				MB_BitStato[100]:=ModBus.MB_MASTER.ReceiveBuffer.Data[3].0; (*Vedi Tabella *)
				MB_BitStato[101]:=ModBus.MB_MASTER.ReceiveBuffer.Data[3].1; (*Vedi Tabella *)
				MB_BitStato[102]:=ModBus.MB_MASTER.ReceiveBuffer.Data[3].2; (*Vedi Tabella *)
				MB_BitStato[103]:=ModBus.MB_MASTER.ReceiveBuffer.Data[3].3; (*Vedi Tabella *)
				MB_BitStato[104]:=ModBus.MB_MASTER.ReceiveBuffer.Data[3].4; (*Vedi Tabella *)
				MB_BitStato[105]:=ModBus.MB_MASTER.ReceiveBuffer.Data[3].5; (*Vedi Tabella *)
				MB_BitStato[106]:=ModBus.MB_MASTER.ReceiveBuffer.Data[3].6; (*Vedi Tabella *)
				MB_BitStato[107]:=ModBus.MB_MASTER.ReceiveBuffer.Data[3].7; (*Vedi Tabella *)
				MB_BitStato[108]:=ModBus.MB_MASTER.ReceiveBuffer.Data[4].0; (*Vedi Tabella *)
				MB_BitStato[109]:=ModBus.MB_MASTER.ReceiveBuffer.Data[4].1; (*Vedi Tabella *)
				MB_BitStato[110]:=ModBus.MB_MASTER.ReceiveBuffer.Data[4].2; (*Vedi Tabella *)
				MB_BitStato[111]:=ModBus.MB_MASTER.ReceiveBuffer.Data[4].3; (*Vedi Tabella *)
				MB_BitStato[112]:=ModBus.MB_MASTER.ReceiveBuffer.Data[4].4; (*Vedi Tabella *)
				MB_BitStato[113]:=ModBus.MB_MASTER.ReceiveBuffer.Data[4].5; (*Vedi Tabella *)
				MB_BitStato[114]:=ModBus.MB_MASTER.ReceiveBuffer.Data[4].6; (*Vedi Tabella *)
				MB_BitStato[115]:=ModBus.MB_MASTER.ReceiveBuffer.Data[4].7; (*Vedi Tabella *)
				MB_BitStato[116]:=ModBus.MB_MASTER.ReceiveBuffer.Data[5].0; (*Vedi Tabella *)
				MB_BitStato[117]:=ModBus.MB_MASTER.ReceiveBuffer.Data[5].1; (*Vedi Tabella *)
				MB_BitStato[118]:=ModBus.MB_MASTER.ReceiveBuffer.Data[5].2; (*Vedi Tabella *)
				MB_BitStato[119]:=ModBus.MB_MASTER.ReceiveBuffer.Data[5].3; (*Vedi Tabella *)
				MB_BitStato[120]:=ModBus.MB_MASTER.ReceiveBuffer.Data[5].4; (*Vedi Tabella *)
				MB_BitStato[121]:=ModBus.MB_MASTER.ReceiveBuffer.Data[5].5; (*Vedi Tabella *)
				MB_BitStato[122]:=ModBus.MB_MASTER.ReceiveBuffer.Data[5].6; (*Vedi Tabella *)
				MB_BitStato[123]:=ModBus.MB_MASTER.ReceiveBuffer.Data[5].7; (*Vedi Tabella *)
				MB_BitStato[124]:=ModBus.MB_MASTER.ReceiveBuffer.Data[6].0; (*Vedi Tabella *)
				MB_BitStato[125]:=ModBus.MB_MASTER.ReceiveBuffer.Data[6].1; (*Vedi Tabella *)
				MB_BitStato[126]:=ModBus.MB_MASTER.ReceiveBuffer.Data[6].2; (*Vedi Tabella *)
				MB_BitStato[127]:=ModBus.MB_MASTER.ReceiveBuffer.Data[6].3; (*Vedi Tabella *)
				MB_BitStato[128]:=ModBus.MB_MASTER.ReceiveBuffer.Data[6].4; (*Vedi Tabella *)
				MB_BitStato[129]:=ModBus.MB_MASTER.ReceiveBuffer.Data[6].5; (*Vedi Tabella *)
				MB_BitStato[130]:=ModBus.MB_MASTER.ReceiveBuffer.Data[6].6; (*Vedi Tabella *)
				MB_BitStato[131]:=ModBus.MB_MASTER.ReceiveBuffer.Data[6].7; (*Vedi Tabella *)
				MB_BitStato[132]:=ModBus.MB_MASTER.ReceiveBuffer.Data[7].0; (*Vedi Tabella *)
				MB_BitStato[133]:=ModBus.MB_MASTER.ReceiveBuffer.Data[7].1; (*Vedi Tabella *)
				MB_BitStato[134]:=ModBus.MB_MASTER.ReceiveBuffer.Data[7].2; (*Vedi Tabella *)
				MB_BitStato[135]:=ModBus.MB_MASTER.ReceiveBuffer.Data[7].3; (*Vedi Tabella *)
				MB_BitStato[136]:=ModBus.MB_MASTER.ReceiveBuffer.Data[7].4; (*Vedi Tabella *)
				MB_BitStato[137]:=ModBus.MB_MASTER.ReceiveBuffer.Data[7].5; (*Vedi Tabella *)
				MB_BitStato[138]:=ModBus.MB_MASTER.ReceiveBuffer.Data[7].6; (*Vedi Tabella *)
				MB_BitStato[139]:=ModBus.MB_MASTER.ReceiveBuffer.Data[7].7; (*Vedi Tabella *)
				MB_BitStato[140]:=ModBus.MB_MASTER.ReceiveBuffer.Data[8].0; (*Vedi Tabella *)
				MB_BitStato[141]:=ModBus.MB_MASTER.ReceiveBuffer.Data[8].1; (*Vedi Tabella *)
				MB_BitStato[142]:=ModBus.MB_MASTER.ReceiveBuffer.Data[8].2; (*Vedi Tabella *)
				MB_BitStato[143]:=ModBus.MB_MASTER.ReceiveBuffer.Data[8].3; (*Vedi Tabella *)
				MB_BitStato[144]:=ModBus.MB_MASTER.ReceiveBuffer.Data[8].4; (*Vedi Tabella *)
				MB_BitStato[145]:=ModBus.MB_MASTER.ReceiveBuffer.Data[8].5; (*Vedi Tabella *)
				MB_BitStato[146]:=ModBus.MB_MASTER.ReceiveBuffer.Data[8].6; (*Vedi Tabella *)
				MB_BitStato[147]:=ModBus.MB_MASTER.ReceiveBuffer.Data[8].7; (*Vedi Tabella *)
				MB_BitStato[148]:=ModBus.MB_MASTER.ReceiveBuffer.Data[9].0; (*Vedi Tabella *)
				MB_BitStato[149]:=ModBus.MB_MASTER.ReceiveBuffer.Data[9].1; (*Vedi Tabella *)
				MB_BitStato[150]:=ModBus.MB_MASTER.ReceiveBuffer.Data[9].2; (*Vedi Tabella *)
				MB_BitStato[151]:=ModBus.MB_MASTER.ReceiveBuffer.Data[9].3; (*Vedi Tabella *)
				MB_BitStato[152]:=ModBus.MB_MASTER.ReceiveBuffer.Data[9].4; (*Vedi Tabella *)
				MB_BitStato[153]:=ModBus.MB_MASTER.ReceiveBuffer.Data[9].5; (*Vedi Tabella *)
				MB_BitStato[154]:=ModBus.MB_MASTER.ReceiveBuffer.Data[9].6; (*Vedi Tabella *)
				MB_BitStato[155]:=ModBus.MB_MASTER.ReceiveBuffer.Data[9].7; (*Vedi Tabella *)
				MB_BitStato[156]:=ModBus.MB_MASTER.ReceiveBuffer.Data[10].0; (*Vedi Tabella *)
				MB_BitStato[157]:=ModBus.MB_MASTER.ReceiveBuffer.Data[10].1; (*Vedi Tabella *)
				MB_BitStato[158]:=ModBus.MB_MASTER.ReceiveBuffer.Data[10].2; (*Vedi Tabella *)
				MB_BitStato[159]:=ModBus.MB_MASTER.ReceiveBuffer.Data[10].3; (*Vedi Tabella *)
				MB_BitStato[160]:=ModBus.MB_MASTER.ReceiveBuffer.Data[10].4; (*Vedi Tabella *)
				MB_BitStato[161]:=ModBus.MB_MASTER.ReceiveBuffer.Data[10].5; (*Vedi Tabella *)
				MB_BitStato[162]:=ModBus.MB_MASTER.ReceiveBuffer.Data[10].6; (*Vedi Tabella *)
				MB_BitStato[163]:=ModBus.MB_MASTER.ReceiveBuffer.Data[10].7; (*Vedi Tabella *)
				MB_BitStato[164]:=ModBus.MB_MASTER.ReceiveBuffer.Data[11].0; (*Vedi Tabella *)
				MB_BitStato[165]:=ModBus.MB_MASTER.ReceiveBuffer.Data[11].1; (*Vedi Tabella *)
				MB_BitStato[166]:=ModBus.MB_MASTER.ReceiveBuffer.Data[11].2; (*Vedi Tabella *)
				MB_BitStato[167]:=ModBus.MB_MASTER.ReceiveBuffer.Data[11].3; (*Vedi Tabella *)
				MB_BitStato[168]:=ModBus.MB_MASTER.ReceiveBuffer.Data[11].4; (*Vedi Tabella *)
				MB_BitStato[169]:=ModBus.MB_MASTER.ReceiveBuffer.Data[11].5; (*Vedi Tabella *)
				MB_BitStato[170]:=ModBus.MB_MASTER.ReceiveBuffer.Data[11].6; (*Vedi Tabella *)
				MB_BitStato[171]:=ModBus.MB_MASTER.ReceiveBuffer.Data[11].7; (*Vedi Tabella *)
				MB_BitStato[172]:=ModBus.MB_MASTER.ReceiveBuffer.Data[12].0; (*Vedi Tabella *)
				MB_BitStato[173]:=ModBus.MB_MASTER.ReceiveBuffer.Data[12].1; (*Vedi Tabella *)
				MB_BitStato[174]:=ModBus.MB_MASTER.ReceiveBuffer.Data[12].2; (*Vedi Tabella *)
				MB_BitStato[175]:=ModBus.MB_MASTER.ReceiveBuffer.Data[12].3; (*Vedi Tabella *)
				MB_BitStato[176]:=ModBus.MB_MASTER.ReceiveBuffer.Data[12].4; (*Vedi Tabella *)
				MB_BitStato[177]:=ModBus.MB_MASTER.ReceiveBuffer.Data[12].5; (*Vedi Tabella *)
				MB_BitStato[178]:=ModBus.MB_MASTER.ReceiveBuffer.Data[12].6; (*Vedi Tabella *)
				MB_BitStato[179]:=ModBus.MB_MASTER.ReceiveBuffer.Data[12].7; (*Vedi Tabella *)
				MB_BitStato[180]:=ModBus.MB_MASTER.ReceiveBuffer.Data[13].0; (*Vedi Tabella *)
				MB_BitStato[181]:=ModBus.MB_MASTER.ReceiveBuffer.Data[13].1; (*Vedi Tabella *)
				MB_BitStato[182]:=ModBus.MB_MASTER.ReceiveBuffer.Data[13].2; (*Vedi Tabella *)
				MB_BitStato[183]:=ModBus.MB_MASTER.ReceiveBuffer.Data[13].3; (*Vedi Tabella *)
				MB_BitStato[184]:=ModBus.MB_MASTER.ReceiveBuffer.Data[13].4; (*Vedi Tabella *)
				MB_BitStato[185]:=ModBus.MB_MASTER.ReceiveBuffer.Data[13].5; (*Vedi Tabella *)
				MB_BitStato[186]:=ModBus.MB_MASTER.ReceiveBuffer.Data[13].6; (*Vedi Tabella *)
				MB_BitStato[187]:=ModBus.MB_MASTER.ReceiveBuffer.Data[13].7; (*Vedi Tabella *)
				MB_BitStato[188]:=ModBus.MB_MASTER.ReceiveBuffer.Data[13].0; (*Vedi Tabella *)
				MB_BitStato[189]:=ModBus.MB_MASTER.ReceiveBuffer.Data[13].1; (*Vedi Tabella *)
				MB_BitStato[190]:=ModBus.MB_MASTER.ReceiveBuffer.Data[13].2; (*Vedi Tabella *)
				MB_BitStato[191]:=ModBus.MB_MASTER.ReceiveBuffer.Data[13].3; (*Vedi Tabella *)
				MB_BitStato[192]:=ModBus.MB_MASTER.ReceiveBuffer.Data[13].4; (*Vedi Tabella *)
				MB_BitStato[193]:=ModBus.MB_MASTER.ReceiveBuffer.Data[13].5; (*Vedi Tabella *)
				MB_BitStato[194]:=ModBus.MB_MASTER.ReceiveBuffer.Data[13].6; (*Vedi Tabella *)
				MB_BitStato[195]:=ModBus.MB_MASTER.ReceiveBuffer.Data[13].7; (*Vedi Tabella *)
				MB_BitStato[196]:=ModBus.MB_MASTER.ReceiveBuffer.Data[14].0; (*Vedi Tabella *)
				MB_BitStato[197]:=ModBus.MB_MASTER.ReceiveBuffer.Data[14].1; (*Vedi Tabella *)
				MB_BitStato[198]:=ModBus.MB_MASTER.ReceiveBuffer.Data[14].2; (*Vedi Tabella *)
				MB_BitStato[199]:=ModBus.MB_MASTER.ReceiveBuffer.Data[14].3; (*Vedi Tabella *)


				state:=290;

			END_IF
		END_IF




		290:    (* Scrittura BOOL - COIL o WORD *)
		IF NOT ModBus.MB_Start THEN
			IF ModBus.MB_MASTER.MB_Error<>0 THEN (*OR ModBus.MB_MASTER.MB_Error<>0 THEN*)
				state := 300;
			ELSE
				IF ScriviDato THEN
					IF ScriviCoil THEN
						Modbus.MB_Query.FunctionCode := 5;
					ELSE
						Modbus.MB_Query.FunctionCode := 6;
					END_IF
					Modbus.MB_Query.SlaveAddress := Address;
					ModBus.MB_Query.Write_StartAddress := IndirizzoDaScrivere;
					ModBus.MB_Query.Write_Quantity :=1;
					ModBus.MB_Query.Write_Data[0] := DatoDaScrivere;
					ModBus.MB_Start := TRUE;
						IF ScriviCoil THEN
							IF 	MB_BitStato[IndirizzoDaScrivere]=WORD_TO_BOOL(DatoDaScrivere-1) THEN
								ScriviDato:=FALSE;
							END_IF
						ELSE
							IF 	MB_RegistriLetti[IndirizzoDaScrivere]=DatoDaScrivere THEN
								ScriviDato:=FALSE;
							END_IF
						END_IF
					state := 295;
				ELSE
					state := 295;
				END_IF
			END_IF
		END_IF




		295:
		IF NOT ModBus.MB_Start THEN
			IF ModBus.MB_MASTER.MB_Error<>0 THEN (*OR ModBus.MB_MASTER.MB_Error<>0 THEN*)
				state := 300;
			ELSE
				IF fModbusAlr THEN fModbusAlr := FALSE; END_IF
				NodoDaInterrogareChiller:=Address+1;
				InibiscoModbusChiller:=FALSE;
				retryErr := 0;
				retry := 0;
				state := 0;
					IF fModbusAlr=FALSE AND ErroreComuModBus=TRUE THEN
						LogEv(EL_Log,EO_CHI,ID,62,'ComunicazioneModBus_OK');
						ErroreComuModBus := FALSE;
				(*	WarningCtr := SEL(WarningCtr=0, WarningCtr-1, 0); *)
					END_IF


			END_IF
		END_IF



	(**** CHECK MODBUS ERROR ****)
	300: 	(* Release MODBUS *)
			InibiscoModbusChiller:=FALSE;
			(* Retries *)
			retry:=retry+1;
			IF retry>3 THEN
				retry:=0;

				(* Verify if slave is dead *)
				IF retryErr < retryErrMaX THEN
					retryErr := retryErr + 1;
				ELSE
					fModbusAlr := TRUE;
					(* Verify ModBus error	*)

					IF fModbusAlr AND ErroreComuModBus=FALSE THEN
						LogEv(EL_Alarm,EO_CHI,ID,61,CONCAT('ErroreModbus_',INT_TO_STRING(ModBus.MB_MASTER.MB_Error)));
						ErroreComuModBus := TRUE;
					END_IF
				END_IF

				END_IF
			Refresh_Now := FALSE;
			NodoDaInterrogareChiller:=Address+1;
			state:=0;
END_CASE




(* Controllo Time Out Ciclo ModBus *)

TimeOutModBus(In:=state<>0,PT:=t#30s);
IF TimeOutModBus.Q THEN
	State:=0;
	Refresh_Now:=TRUE;  (* Rilancio la lettura del nodo *)
	IF MODBUS.MB_Lock=TRUE THEN MODBUS.MB_Lock:=FALSE;END_IF
	IF InibiscoModbusChiller=TRUE THEN InibiscoModbusChiller:=FALSE;END_IF
END_IF
END_ACTION

(* POU Utils Functions/TONOF, ST *)
FUNCTION_BLOCK TONOF
VAR_INPUT
	IN		: BOOL;
	PT_ON	: TIME; (* time to pass, before OUT is set *)
	PT_OF	: TIME; (* time to pass, before OUT is reset *)
END_VAR
VAR_OUTPUT
	OUT		: BOOL;
END_VAR
VAR
	timer	: TON;
END_VAR
IF IN<>OUT THEN
	timer(IN:=TRUE,PT:=SEL(IN,PT_OF,PT_ON));
	IF timer.Q THEN OUT:=IN; END_IF
ELSE
	timer(IN:=FALSE);
END_IF
END_FUNCTION_BLOCK

(* POU Plant_Objects/obj_MODBUS_TRENDCOIN_01, ST *)
FUNCTION_BLOCK obj_MODBUS_TRENDCOIN_01
VAR CONSTANT

	TimeOutModBus: TON;


END_VAR
VAR_INPUT
	ID			:	BYTE;
	Address		:	BYTE;
	(* Modbus *)
	Refresh_Now	:	BOOL;			(* Richiesta di lettura stato macchina Immediata  *)
	retryErrMax	:	BYTE := 2;

	IndirizzoDaScrivere: WORD;
	DatoDaScrivere: INT;
	ScriviDato: BOOL;
	ScriviCoil: BOOL;

(* Variabili da scrivere nel parametri Trend *)

(*	EnScrittura		:ARRAY [0..15] OF	FLT_EVENT; *)

	ControlMode_UTA01:BOOL;     (* 0 = controllato in manuale ; 1 = controllato col Crono *)
	ControlMode_UTA02:BOOL;
	ControlMode_UTA03:BOOL;
	ControlMode_UTA04:BOOL;
	ControlMode_UTA05:BOOL;
	ControlMode_UTA06:BOOL;
	ControlMode_UTA07:BOOL;
	ControlMode_UTA08:BOOL;
	ControlMode_UTA09:BOOL;
	ControlMode_UTA10:BOOL;
	ControlMode_UTA12:BOOL;
	ControlMode_UTA13:BOOL;

	ScriviRUN_UTA01:BOOL;
	ScriviRUN_UTA02:BOOL;
	ScriviRUN_UTA03:BOOL;
	ScriviRUN_UTA04:BOOL;
	ScriviRUN_UTA05:BOOL;
	ScriviRUN_UTA06:BOOL;
	ScriviRUN_UTA07:BOOL;
	ScriviRUN_UTA08:BOOL;
	ScriviRUN_UTA09:BOOL;
	ScriviRUN_UTA10:BOOL;
	ScriviRUN_UTA12:BOOL;
	ScriviRUN_UTA13:BOOL;

	ScriviSP_UTA01:INT;
	ScriviSP_UTA02:INT;
	ScriviSP_UTA03:INT;
	ScriviSP_UTA04:INT;
	ScriviSP_UTA05:INT;
	ScriviSP_UTA06:INT;
	ScriviSP_UTA07:INT;
	ScriviSP_UTA08:INT;
	ScriviSP_UTA09:INT;
	ScriviSP_UTA10:INT;
	ScriviSP_UTA12:INT;
	ScriviSP_UTA13:INT;


END_VAR
VAR_IN_OUT
	ModBus		:obj_MODBUS;

END_VAR
VAR_OUTPUT
	Status_Log	:	WORD;
	Status_Vis	:	DWORD;
END_VAR
VAR

	state		:	INT;
	retry		:	BYTE;
	retryErr	:	BYTE;
	ReadTmr		:	TON := (PT:=T#5s);
	fModbusAlr:BOOL;

(*	retry_write	:	BYTE;
	fWriteStatus:	BOOL;
	fWriteMode	:	BOOL;
	fWriteReset	:	BOOL; *)

	x: INT;

	VerificaFuctionCode: INT;
	VerificaNodoLetto: INT;
	ErroreComuModBus: BOOL;
	IndiceErrore: BYTE;

	MB_BitStato: ARRAY [0..450] OF BOOL;
	MB_RegistriLetti: ARRAY [0..450] OF INT;
	MB_RegistriHoldingLetti: ARRAY [0..170] OF INT;
	MB_BitStatoCoil: ARRAY [0..100] OF BOOL;




	AddressRead: BYTE;
	index: BYTE;
	indexErr: BYTE;


	Read_StartAddress: INT;
	Read_Quantity: BYTE;
	IndiceMBLettura: INT;
	IndiceMBLetto: INT;



	test_Address: INT;
	Test_ScriviCoil: BOOL;
	test_Write: WORD;
	ScriviMB: BOOL;



	AddressDaScrivere: INT;


	temp :STRING(255);
	tempRaw		: ARRAY [0..MAX_SEND_TCP_CLIENT] OF BYTE;
	tempRawLen :DINT;
	longString:STRING(800);


END_VAR
(*
	EnScrittura[1](IN:=Abilita_UTA01);
	ScriviRUN_UTA01:=EnScrittura[1].EVH;
	ScriviRUN_UTA01:=EnScrittura[1].EVL;

	EnScrittura[2](IN:=Abilita_UTA02);
	ScriviRUN_UTA02:=EnScrittura[2].EVH;
	ScriviRUN_UTA02:=EnScrittura[2].EVL;

	EnScrittura[3](IN:=Abilita_UTA03);
	ScriviRUN_UTA03:=EnScrittura[3].EVH;
	ScriviRUN_UTA03:=EnScrittura[3].EVL;

	EnScrittura[4](IN:=Abilita_UTA04);
	ScriviRUN_UTA04:=EnScrittura[4].EVH;
	ScriviRUN_UTA04:=EnScrittura[4].EVL;

	EnScrittura[4](IN:=Abilita_UTA04);
	ScriviRUN_UTA04:=EnScrittura[4].EVH;
	ScriviRUN_UTA04:=EnScrittura[4].EVL;

	EnScrittura[5](IN:=Abilita_UTA05);
	ScriviRUN_UTA05:=EnScrittura[5].EVH;
	ScriviRUN_UTA05:=EnScrittura[5].EVL;

	EnScrittura[6](IN:=Abilita_UTA06);
	ScriviRUN_UTA06:=EnScrittura[6].EVH;
	ScriviRUN_UTA06:=EnScrittura[6].EVL;

	EnScrittura[7](IN:=Abilita_UTA07);
	ScriviRUN_UTA07:=EnScrittura[7].EVH;
	ScriviRUN_UTA07:=EnScrittura[7].EVL;

	EnScrittura[8](IN:=Abilita_UTA08);
	ScriviRUN_UTA08:=EnScrittura[8].EVH;
	ScriviRUN_UTA08:=EnScrittura[8].EVL;

	EnScrittura[9](IN:=Abilita_UTA09);
	ScriviRUN_UTA09:=EnScrittura[9].EVH;
	ScriviRUN_UTA09:=EnScrittura[9].EVL;

	EnScrittura[10](IN:=Abilita_UTA10);
	ScriviRUN_UTA10:=EnScrittura[10].EVH;
	ScriviRUN_UTA10:=EnScrittura[10].EVL;

(*	EnScrittura[11](IN:=Abilita_UTA11);
	ScriviRUN_UTA11:=EnScrittura[11].EVH;
	ScriviRUN_UTA11:=EnScrittura[11].EVL; *)

	EnScrittura[12](IN:=Abilita_UTA12);
	ScriviRUN_UTA12:=EnScrittura[12].EVH;
	ScriviRUN_UTA12:=EnScrittura[12].EVL;

	EnScrittura[13](IN:=Abilita_UTA13);
	ScriviRUN_UTA13:=EnScrittura[13].EVH;
	ScriviRUN_UTA13:=EnScrittura[13].EVL;
*)





(* Call ModBus state machine *)
Stm();

(* Check alarm	*)




(* Seganalzione stato Frigorifero  *)
IF ErroreComuModBus THEN
		Status_Log:=2; Status_Vis:=16#2020F0;
(*	ELSIF Warning OR Warning2 THEN
		Status_Log:=1; Status_Vis:=16#20F0F0; *)
    ELSE
		Status_Log:=0;
		Status_Vis:=16#006000;
END_IF
END_FUNCTION_BLOCK
ACTION AddLogData:
Logger.s1:=INSERT('&POOL=',BYTE_TO_STRING(ID),5);
IF ID<10 THEN Logger.s1:=INSERT(Logger.s1,'0',5); END_IF


(* inizializzo stringa da loggare **)
FOR tempRawLen:=0 TO MAX_SEND_TCP_CLIENT DO
                tempRaw[tempRawLen]:=0;
END_FOR

tempRawLen:=0;


temp:=Logger.s1;
ADDSTRING(ADR(tempRaw), ADR(temp), tempRawLen);

(* Sparo i COIL **)
FOR x:= 1 TO 65 DO
	temp:=CONCAT(SEL(MB_BitStatoCoil[x],'0','1'),';');
	ADDSTRING(ADR(tempRaw), ADR(temp), tempRawLen);
END_FOR

(* Sparo gli ingressi Digitali **)
FOR x:= 1 TO 358 DO
	temp:=CONCAT(SEL(MB_BitStato[x],'0','1'),';');
	ADDSTRING(ADR(tempRaw), ADR(temp), tempRawLen);
END_FOR

(* Sparo gli HOLDING **)
FOR x:= 1 TO 168 DO
	temp:=CONCAT(INT_TO_STRING(MB_RegistriHoldingLetti[x]),';');
	ADDSTRING(ADR(tempRaw), ADR(temp), tempRawLen);
END_FOR

(* Sparo gli integer **)
FOR x:= 1 TO 283 DO
	temp:=CONCAT(INT_TO_STRING(MB_RegistriLetti[x]),';');
	ADDSTRING(ADR(tempRaw), ADR(temp), tempRawLen);
END_FOR

	temp:=(INT_TO_STRING(MB_RegistriLetti[284]));
	ADDSTRING(ADR(tempRaw), ADR(temp), tempRawLen);

ADDSTRING(ADR(Logger.TData), ADR(tempRaw), Logger.TLen);
END_ACTION
ACTION Stm:
CASE state OF
	0:	(* Refresh time manager *)
		ReadTmr(IN:=NOT ReadTmr.Q);
		(*A tempo interrogo il nodo sempre che non ci sia qualcuno che lo sta interrogando in quel momento *)

		IF (ReadTmr.Q AND NodoDaInterrogareMB1=Address )OR Refresh_Now AND NOT InibiscoModbusMB1 THEN
			state := 10;
			ReadTmr.PT := T#10s;  (* moreno *)
			Refresh_Now := FALSE;
			InibiscoModbusMB1 := TRUE;
		END_IF

	(**** Leggo le Analogiche a Disposzione  ****)

	10:	(* richiedo lettura di tutti gli Input Register   *)

		Modbus.MB_Query.SlaveAddress := Address;
		Modbus.MB_Query.FunctionCode := 4;
		Read_StartAddress := 0 ;			(* richiedo lettura altri Parametri *)
		Read_Quantity := 20;
		ModBus.MB_Start := TRUE;
		state := 20;


	20:
		ModBus.MB_Query.Read_StartAddress := 0 ;			(* richiedo lettura altri Parametri *)
		ModBus.MB_Query.Read_Quantity := 20;
		ModBus.MB_Start := TRUE;
		Read_StartAddress := 0 ;
		state := 30;



	30:	(* Risposta all'interrogazione *)
		IF NOT ModBus.MB_Start   THEN
			VerificaFuctionCode:=ModBus.MB_Resp.FunctionCode;
			VerificaNodoLetto:=ModBus.MB_Resp.SlaveAddress;

			IF ModBus.MB_MASTER.MB_Error<>0 THEN
				state := 300;
			ELSE

				FOR x:= 0 TO ModBus.MB_Query.Read_Quantity DO
					MB_RegistriLetti[Read_StartAddress+x ] := ModBus.MB_Resp.Data[x];   	(* Vedi tabella *)
				END_FOR

			ModBus.MB_Query.Read_StartAddress := 20 ;			(* richiedo lettura altri Parametri *)
			ModBus.MB_Query.Read_Quantity := 20;
			ModBus.MB_Start := TRUE;
			Read_StartAddress := 20 ;
			state := 31;
			END_IF
		END_IF


	31:	(* Risposta all'interrogazione *)
		IF NOT ModBus.MB_Start   THEN
			VerificaFuctionCode:=ModBus.MB_Resp.FunctionCode;
			VerificaNodoLetto:=ModBus.MB_Resp.SlaveAddress;

			IF ModBus.MB_MASTER.MB_Error<>0 THEN
				state := 300;
			ELSE

				FOR x:= 0 TO ModBus.MB_Query.Read_Quantity DO
					MB_RegistriLetti[Read_StartAddress+x ] := ModBus.MB_Resp.Data[x];   	(* Vedi tabella *)
				END_FOR

			ModBus.MB_Query.Read_StartAddress := 40 ;			(* richiedo lettura altri Parametri *)
			ModBus.MB_Query.Read_Quantity := 20;
			ModBus.MB_Start := TRUE;
			Read_StartAddress := 40 ;
			state := 32;
			END_IF
		END_IF



	32:	(* Risposta all'interrogazione *)
		IF NOT ModBus.MB_Start   THEN
			VerificaFuctionCode:=ModBus.MB_Resp.FunctionCode;
			VerificaNodoLetto:=ModBus.MB_Resp.SlaveAddress;

			IF ModBus.MB_MASTER.MB_Error<>0 THEN
				state := 300;
			ELSE

				FOR x:= 0 TO ModBus.MB_Query.Read_Quantity DO
					MB_RegistriLetti[Read_StartAddress+x ] := ModBus.MB_Resp.Data[x];   	(* Vedi tabella *)
				END_FOR

			ModBus.MB_Query.Read_StartAddress := 60 ;			(* richiedo lettura altri Parametri *)
			ModBus.MB_Query.Read_Quantity := 20;
			ModBus.MB_Start := TRUE;
			Read_StartAddress := 60 ;
			state := 33;
			END_IF
		END_IF

	33:	(* Risposta all'interrogazione *)
		IF NOT ModBus.MB_Start   THEN
			VerificaFuctionCode:=ModBus.MB_Resp.FunctionCode;
			VerificaNodoLetto:=ModBus.MB_Resp.SlaveAddress;

			IF ModBus.MB_MASTER.MB_Error<>0 THEN
				state := 300;
			ELSE

				FOR x:= 0 TO ModBus.MB_Query.Read_Quantity DO
					MB_RegistriLetti[Read_StartAddress+x ] := ModBus.MB_Resp.Data[x];   	(* Vedi tabella *)
				END_FOR

			ModBus.MB_Query.Read_StartAddress := 80 ;			(* richiedo lettura altri Parametri *)
			ModBus.MB_Query.Read_Quantity := 20;
			ModBus.MB_Start := TRUE;
			Read_StartAddress := 80 ;
			state := 34;
			END_IF
		END_IF


	34:	(* Risposta all'interrogazione *)
		IF NOT ModBus.MB_Start   THEN
			VerificaFuctionCode:=ModBus.MB_Resp.FunctionCode;
			VerificaNodoLetto:=ModBus.MB_Resp.SlaveAddress;

			IF ModBus.MB_MASTER.MB_Error<>0 THEN
				state := 300;
			ELSE

				FOR x:= 0 TO ModBus.MB_Query.Read_Quantity DO
					MB_RegistriLetti[Read_StartAddress+x ] := ModBus.MB_Resp.Data[x];   	(* Vedi tabella *)
				END_FOR

			ModBus.MB_Query.Read_StartAddress := 100 ;			(* richiedo lettura altri Parametri *)
			ModBus.MB_Query.Read_Quantity := 20;
			ModBus.MB_Start := TRUE;
			Read_StartAddress := 100 ;
			state := 35;
			END_IF
		END_IF


	35:	(* Risposta all'interrogazione *)
		IF NOT ModBus.MB_Start   THEN
			VerificaFuctionCode:=ModBus.MB_Resp.FunctionCode;
			VerificaNodoLetto:=ModBus.MB_Resp.SlaveAddress;

			IF ModBus.MB_MASTER.MB_Error<>0 THEN
				state := 300;
			ELSE

				FOR x:= 0 TO ModBus.MB_Query.Read_Quantity DO
					MB_RegistriLetti[Read_StartAddress+x ] := ModBus.MB_Resp.Data[x];   	(* Vedi tabella *)
				END_FOR

			ModBus.MB_Query.Read_StartAddress := 120 ;			(* richiedo lettura altri Parametri *)
			ModBus.MB_Query.Read_Quantity := 20;
			ModBus.MB_Start := TRUE;
			Read_StartAddress := 120 ;
			state := 36;
			END_IF
		END_IF

	36:	(* Risposta all'interrogazione *)
		IF NOT ModBus.MB_Start   THEN
			VerificaFuctionCode:=ModBus.MB_Resp.FunctionCode;
			VerificaNodoLetto:=ModBus.MB_Resp.SlaveAddress;

			IF ModBus.MB_MASTER.MB_Error<>0 THEN
				state := 300;
			ELSE

				FOR x:= 0 TO ModBus.MB_Query.Read_Quantity DO
					MB_RegistriLetti[Read_StartAddress+x ] := ModBus.MB_Resp.Data[x];   	(* Vedi tabella *)
				END_FOR

			ModBus.MB_Query.Read_StartAddress := 140 ;			(* richiedo lettura altri Parametri *)
			ModBus.MB_Query.Read_Quantity := 20;
			ModBus.MB_Start := TRUE;
			Read_StartAddress := 140 ;
			state := 37;
			END_IF
		END_IF

	37:	(* Risposta all'interrogazione *)
		IF NOT ModBus.MB_Start   THEN
			VerificaFuctionCode:=ModBus.MB_Resp.FunctionCode;
			VerificaNodoLetto:=ModBus.MB_Resp.SlaveAddress;

			IF ModBus.MB_MASTER.MB_Error<>0 THEN
				state := 300;
			ELSE

				FOR x:= 0 TO ModBus.MB_Query.Read_Quantity DO
					MB_RegistriLetti[Read_StartAddress+x ] := ModBus.MB_Resp.Data[x];   	(* Vedi tabella *)
				END_FOR

			ModBus.MB_Query.Read_StartAddress := 160 ;			(* richiedo lettura altri Parametri *)
			ModBus.MB_Query.Read_Quantity := 20;
			ModBus.MB_Start := TRUE;
			Read_StartAddress := 160 ;
			state := 38;
			END_IF
		END_IF

	38:	(* Risposta all'interrogazione *)
		IF NOT ModBus.MB_Start   THEN
			VerificaFuctionCode:=ModBus.MB_Resp.FunctionCode;
			VerificaNodoLetto:=ModBus.MB_Resp.SlaveAddress;

			IF ModBus.MB_MASTER.MB_Error<>0 THEN
				state := 300;
			ELSE

				FOR x:= 0 TO ModBus.MB_Query.Read_Quantity DO
					MB_RegistriLetti[Read_StartAddress+x ] := ModBus.MB_Resp.Data[x];   	(* Vedi tabella *)
				END_FOR

			ModBus.MB_Query.Read_StartAddress := 180 ;			(* richiedo lettura altri Parametri *)
			ModBus.MB_Query.Read_Quantity := 20;
			ModBus.MB_Start := TRUE;
			Read_StartAddress := 180 ;
			state := 39;
			END_IF
		END_IF

	39:	(* Risposta all'interrogazione *)
		IF NOT ModBus.MB_Start   THEN
			VerificaFuctionCode:=ModBus.MB_Resp.FunctionCode;
			VerificaNodoLetto:=ModBus.MB_Resp.SlaveAddress;

			IF ModBus.MB_MASTER.MB_Error<>0 THEN
				state := 300;
			ELSE

				FOR x:= 0 TO ModBus.MB_Query.Read_Quantity DO
					MB_RegistriLetti[Read_StartAddress+x ] := ModBus.MB_Resp.Data[x];   	(* Vedi tabella *)
				END_FOR

			ModBus.MB_Query.Read_StartAddress := 200 ;			(* richiedo lettura altri Parametri *)
			ModBus.MB_Query.Read_Quantity := 20;
			ModBus.MB_Start := TRUE;
			Read_StartAddress := 200 ;
			state := 40;
			END_IF
		END_IF

	40:	(* Risposta all'interrogazione *)
		IF NOT ModBus.MB_Start   THEN
			VerificaFuctionCode:=ModBus.MB_Resp.FunctionCode;
			VerificaNodoLetto:=ModBus.MB_Resp.SlaveAddress;

			IF ModBus.MB_MASTER.MB_Error<>0 THEN
				state := 300;
			ELSE

				FOR x:= 0 TO ModBus.MB_Query.Read_Quantity DO
					MB_RegistriLetti[Read_StartAddress+x ] := ModBus.MB_Resp.Data[x];   	(* Vedi tabella *)
				END_FOR

			ModBus.MB_Query.Read_StartAddress := 220 ;			(* richiedo lettura altri Parametri *)
			ModBus.MB_Query.Read_Quantity := 20;
			ModBus.MB_Start := TRUE;
			Read_StartAddress := 220 ;
			state := 41;
			END_IF
		END_IF

	41:	(* Risposta all'interrogazione *)
		IF NOT ModBus.MB_Start   THEN
			VerificaFuctionCode:=ModBus.MB_Resp.FunctionCode;
			VerificaNodoLetto:=ModBus.MB_Resp.SlaveAddress;

			IF ModBus.MB_MASTER.MB_Error<>0 THEN
				state := 300;
			ELSE

				FOR x:= 0 TO ModBus.MB_Query.Read_Quantity DO
					MB_RegistriLetti[Read_StartAddress+x ] := ModBus.MB_Resp.Data[x];   	(* Vedi tabella *)
				END_FOR

			ModBus.MB_Query.Read_StartAddress := 240 ;			(* richiedo lettura altri Parametri *)
			ModBus.MB_Query.Read_Quantity := 20;
			ModBus.MB_Start := TRUE;
			Read_StartAddress := 240 ;
			state := 42;
			END_IF
		END_IF

	42:	(* Risposta all'interrogazione *)
		IF NOT ModBus.MB_Start   THEN
			VerificaFuctionCode:=ModBus.MB_Resp.FunctionCode;
			VerificaNodoLetto:=ModBus.MB_Resp.SlaveAddress;

			IF ModBus.MB_MASTER.MB_Error<>0 THEN
				state := 300;
			ELSE

				FOR x:= 0 TO ModBus.MB_Query.Read_Quantity DO
					MB_RegistriLetti[Read_StartAddress+x ] := ModBus.MB_Resp.Data[x];   	(* Vedi tabella *)
				END_FOR

			ModBus.MB_Query.Read_StartAddress := 260 ;			(* richiedo lettura altri Parametri *)
			ModBus.MB_Query.Read_Quantity := 20;
			ModBus.MB_Start := TRUE;
			Read_StartAddress := 260 ;
			state := 43;
			END_IF
		END_IF

	43:	(* Risposta all'interrogazione *)
		IF NOT ModBus.MB_Start   THEN
			VerificaFuctionCode:=ModBus.MB_Resp.FunctionCode;
			VerificaNodoLetto:=ModBus.MB_Resp.SlaveAddress;

			IF ModBus.MB_MASTER.MB_Error<>0 THEN
				state := 300;
			ELSE

				FOR x:= 0 TO ModBus.MB_Query.Read_Quantity DO
					MB_RegistriLetti[Read_StartAddress+x ] := ModBus.MB_Resp.Data[x];   	(* Vedi tabella *)
				END_FOR

			ModBus.MB_Query.Read_StartAddress := 280 ;			(* richiedo lettura altri Parametri *)
			ModBus.MB_Query.Read_Quantity := 4;
			ModBus.MB_Start := TRUE;
			Read_StartAddress := 280 ;
			state := 44;
			END_IF
		END_IF

	44:	(* Risposta all'interrogazione *)
		IF NOT ModBus.MB_Start   THEN
			VerificaFuctionCode:=ModBus.MB_Resp.FunctionCode;
			VerificaNodoLetto:=ModBus.MB_Resp.SlaveAddress;

			IF ModBus.MB_MASTER.MB_Error<>0 THEN
				state := 300;
			ELSE

				FOR x:= 0 TO ModBus.MB_Query.Read_Quantity DO
					MB_RegistriLetti[Read_StartAddress+x ] := ModBus.MB_Resp.Data[x];   	(* Vedi tabella *)
				END_FOR

		(*	ModBus.MB_Query.Read_StartAddress := 280 ;			(* richiedo lettura altri Parametri *)
			ModBus.MB_Query.Read_Quantity := 4;
			ModBus.MB_Start := TRUE;
			Read_StartAddress := 280 ; *)
			state := 50;
			END_IF
		END_IF





	50:	(* Risposta all'interrogazione Holding*)

		Modbus.MB_Query.FunctionCode := 3;
		Read_StartAddress := 0 ;			(* richiedo lettura altri Parametri *)
		Read_Quantity := 20;
		ModBus.MB_Start := TRUE;
		state := 51;

	51:	(* Risposta all'interrogazione *)
		IF NOT ModBus.MB_Start   THEN
			VerificaFuctionCode:=ModBus.MB_Resp.FunctionCode;
			VerificaNodoLetto:=ModBus.MB_Resp.SlaveAddress;

			IF ModBus.MB_MASTER.MB_Error<>0 THEN
				state := 300;
			ELSE

				FOR x:= 0 TO ModBus.MB_Query.Read_Quantity DO
					MB_RegistriHoldingLetti[Read_StartAddress+x ] := ModBus.MB_Resp.Data[x];   	(* Vedi tabella *)
				END_FOR

			ModBus.MB_Query.Read_StartAddress := 0 ;			(* richiedo lettura altri Parametri *)
			ModBus.MB_Query.Read_Quantity := 20;
			ModBus.MB_Start := TRUE;
			Read_StartAddress := 0 ;
			state := 511;
			END_IF
		END_IF


	511:	(* Risposta all'interrogazione *)
		IF NOT ModBus.MB_Start   THEN
			VerificaFuctionCode:=ModBus.MB_Resp.FunctionCode;
			VerificaNodoLetto:=ModBus.MB_Resp.SlaveAddress;

			IF ModBus.MB_MASTER.MB_Error<>0 THEN
				state := 300;
			ELSE

				FOR x:= 0 TO ModBus.MB_Query.Read_Quantity DO
					MB_RegistriHoldingLetti[Read_StartAddress+x ] := ModBus.MB_Resp.Data[x];   	(* Vedi tabella *)
				END_FOR

			ModBus.MB_Query.Read_StartAddress := 20 ;			(* richiedo lettura altri Parametri *)
			ModBus.MB_Query.Read_Quantity := 20;
			ModBus.MB_Start := TRUE;
			Read_StartAddress := 20 ;
			state := 52;
			END_IF
		END_IF

	52:	(* Risposta all'interrogazione *)
		IF NOT ModBus.MB_Start   THEN
			VerificaFuctionCode:=ModBus.MB_Resp.FunctionCode;
			VerificaNodoLetto:=ModBus.MB_Resp.SlaveAddress;

			IF ModBus.MB_MASTER.MB_Error<>0 THEN
				state := 300;
			ELSE

				FOR x:= 0 TO ModBus.MB_Query.Read_Quantity DO
					MB_RegistriHoldingLetti[Read_StartAddress+x ] := ModBus.MB_Resp.Data[x];   	(* Vedi tabella *)
				END_FOR

			ModBus.MB_Query.Read_StartAddress := 40 ;			(* richiedo lettura altri Parametri *)
			ModBus.MB_Query.Read_Quantity := 20;
			ModBus.MB_Start := TRUE;
			Read_StartAddress := 40 ;
			state := 53;
			END_IF
		END_IF

	53:	(* Risposta all'interrogazione *)
		IF NOT ModBus.MB_Start   THEN
			VerificaFuctionCode:=ModBus.MB_Resp.FunctionCode;
			VerificaNodoLetto:=ModBus.MB_Resp.SlaveAddress;

			IF ModBus.MB_MASTER.MB_Error<>0 THEN
				state := 300;
			ELSE

				FOR x:= 0 TO ModBus.MB_Query.Read_Quantity DO
					MB_RegistriHoldingLetti[Read_StartAddress+x ] := ModBus.MB_Resp.Data[x];   	(* Vedi tabella *)
				END_FOR

			ModBus.MB_Query.Read_StartAddress := 60 ;			(* richiedo lettura altri Parametri *)
			ModBus.MB_Query.Read_Quantity := 20;
			ModBus.MB_Start := TRUE;
			Read_StartAddress := 60 ;
			state := 54;
			END_IF
		END_IF

	54:	(* Risposta all'interrogazione *)
		IF NOT ModBus.MB_Start   THEN
			VerificaFuctionCode:=ModBus.MB_Resp.FunctionCode;
			VerificaNodoLetto:=ModBus.MB_Resp.SlaveAddress;

			IF ModBus.MB_MASTER.MB_Error<>0 THEN
				state := 300;
			ELSE

				FOR x:= 0 TO ModBus.MB_Query.Read_Quantity DO
					MB_RegistriHoldingLetti[Read_StartAddress+x ] := ModBus.MB_Resp.Data[x];   	(* Vedi tabella *)
				END_FOR

			ModBus.MB_Query.Read_StartAddress := 80 ;			(* richiedo lettura altri Parametri *)
			ModBus.MB_Query.Read_Quantity := 20;
			ModBus.MB_Start := TRUE;
			Read_StartAddress := 80 ;
			state := 55;
			END_IF
		END_IF

	55:	(* Risposta all'interrogazione *)
		IF NOT ModBus.MB_Start   THEN
			VerificaFuctionCode:=ModBus.MB_Resp.FunctionCode;
			VerificaNodoLetto:=ModBus.MB_Resp.SlaveAddress;

			IF ModBus.MB_MASTER.MB_Error<>0 THEN
				state := 300;
			ELSE

				FOR x:= 0 TO ModBus.MB_Query.Read_Quantity DO
					MB_RegistriHoldingLetti[Read_StartAddress+x ] := ModBus.MB_Resp.Data[x];   	(* Vedi tabella *)
				END_FOR

			ModBus.MB_Query.Read_StartAddress := 100 ;			(* richiedo lettura altri Parametri *)
			ModBus.MB_Query.Read_Quantity := 20;
			ModBus.MB_Start := TRUE;
			Read_StartAddress := 100 ;
			state := 56;
			END_IF
		END_IF

	56:	(* Risposta all'interrogazione *)
		IF NOT ModBus.MB_Start   THEN
			VerificaFuctionCode:=ModBus.MB_Resp.FunctionCode;
			VerificaNodoLetto:=ModBus.MB_Resp.SlaveAddress;

			IF ModBus.MB_MASTER.MB_Error<>0 THEN
				state := 300;
			ELSE

				FOR x:= 0 TO ModBus.MB_Query.Read_Quantity DO
					MB_RegistriHoldingLetti[Read_StartAddress+x ] := ModBus.MB_Resp.Data[x];   	(* Vedi tabella *)
				END_FOR

			ModBus.MB_Query.Read_StartAddress := 120 ;			(* richiedo lettura altri Parametri *)
			ModBus.MB_Query.Read_Quantity := 20;
			ModBus.MB_Start := TRUE;
			Read_StartAddress := 120 ;
			state := 57;
			END_IF
		END_IF

	57:	(* Risposta all'interrogazione *)
		IF NOT ModBus.MB_Start   THEN
			VerificaFuctionCode:=ModBus.MB_Resp.FunctionCode;
			VerificaNodoLetto:=ModBus.MB_Resp.SlaveAddress;

			IF ModBus.MB_MASTER.MB_Error<>0 THEN
				state := 300;
			ELSE

				FOR x:= 0 TO ModBus.MB_Query.Read_Quantity DO
					MB_RegistriHoldingLetti[Read_StartAddress+x ] := ModBus.MB_Resp.Data[x];   	(* Vedi tabella *)
				END_FOR

			ModBus.MB_Query.Read_StartAddress := 140 ;			(* richiedo lettura altri Parametri *)
			ModBus.MB_Query.Read_Quantity := 20;
			ModBus.MB_Start := TRUE;
			Read_StartAddress := 140 ;
			state := 58;
			END_IF
		END_IF

	58:	(* Risposta all'interrogazione *)
		IF NOT ModBus.MB_Start   THEN
			VerificaFuctionCode:=ModBus.MB_Resp.FunctionCode;
			VerificaNodoLetto:=ModBus.MB_Resp.SlaveAddress;

			IF ModBus.MB_MASTER.MB_Error<>0 THEN
				state := 300;
			ELSE

				FOR x:= 0 TO ModBus.MB_Query.Read_Quantity DO
					MB_RegistriHoldingLetti[Read_StartAddress+x ] := ModBus.MB_Resp.Data[x];   	(* Vedi tabella *)
				END_FOR

			ModBus.MB_Query.Read_StartAddress := 160 ;			(* richiedo lettura altri Parametri *)
			ModBus.MB_Query.Read_Quantity := 8;
			ModBus.MB_Start := TRUE;
			Read_StartAddress := 160 ;
			state := 59;
			END_IF
		END_IF

	59:	(* Risposta all'interrogazione *)
		IF NOT ModBus.MB_Start   THEN
			VerificaFuctionCode:=ModBus.MB_Resp.FunctionCode;
			VerificaNodoLetto:=ModBus.MB_Resp.SlaveAddress;

			IF ModBus.MB_MASTER.MB_Error<>0 THEN
				state := 300;
			ELSE

				FOR x:= 0 TO ModBus.MB_Query.Read_Quantity DO
					MB_RegistriHoldingLetti[Read_StartAddress+x ] := ModBus.MB_Resp.Data[x];   	(* Vedi tabella *)
				END_FOR

		(*	ModBus.MB_Query.Read_StartAddress := 160 ;			(* richiedo lettura altri Parametri *)
			ModBus.MB_Query.Read_Quantity := 20;
			ModBus.MB_Start := TRUE;
			Read_StartAddress := 160 ; *)
			state := 100;
			END_IF
		END_IF





	100: (* Rispota Altri paramenti Digital Input *)
		IF NOT ModBus.MB_Start  THEN

			IF ModBus.MB_MASTER.MB_Error<>0 THEN
				state := 300;
			ELSE
				Modbus.MB_Query.SlaveAddress := Address;
				Modbus.MB_Query.FunctionCode := 2;
				ModBus.MB_Query.Read_StartAddress := 0;	(* richiedo lettura altri Parametri *)
				ModBus.MB_Query.Read_Quantity := 64;
				ModBus.MB_Start := TRUE;

				state:=105;
			END_IF
		END_IF
	105: (* Rispota Altri paramenti *)

		IF NOT ModBus.MB_Start  THEN

			IF ModBus.MB_MASTER.MB_Error<>0 THEN
				state := 300;
			ELSE

				MB_BitStato[0]:=ModBus.MB_MASTER.ReceiveBuffer.Data[3].0; (*Vedi Tabella *)
				MB_BitStato[1]:=ModBus.MB_MASTER.ReceiveBuffer.Data[3].1; (*Vedi Tabella *)
				MB_BitStato[2]:=ModBus.MB_MASTER.ReceiveBuffer.Data[3].2; (*Vedi Tabella *)
				MB_BitStato[3]:=ModBus.MB_MASTER.ReceiveBuffer.Data[3].3; (*Vedi Tabella *)
				MB_BitStato[4]:=ModBus.MB_MASTER.ReceiveBuffer.Data[3].4; (*Vedi Tabella *)
				MB_BitStato[5]:=ModBus.MB_MASTER.ReceiveBuffer.Data[3].5; (*Vedi Tabella *)
				MB_BitStato[6]:=ModBus.MB_MASTER.ReceiveBuffer.Data[3].6; (*Vedi Tabella *)
				MB_BitStato[7]:=ModBus.MB_MASTER.ReceiveBuffer.Data[3].7; (*Vedi Tabella *)
				MB_BitStato[8]:=ModBus.MB_MASTER.ReceiveBuffer.Data[4].0; (*Vedi Tabella *)
				MB_BitStato[9]:=ModBus.MB_MASTER.ReceiveBuffer.Data[4].1; (*Vedi Tabella *)
				MB_BitStato[10]:=ModBus.MB_MASTER.ReceiveBuffer.Data[4].2; (*Vedi Tabella *)
				MB_BitStato[11]:=ModBus.MB_MASTER.ReceiveBuffer.Data[4].3; (*Vedi Tabella *)
				MB_BitStato[12]:=ModBus.MB_MASTER.ReceiveBuffer.Data[4].4; (*Vedi Tabella *)
				MB_BitStato[13]:=ModBus.MB_MASTER.ReceiveBuffer.Data[4].5; (*Vedi Tabella *)
				MB_BitStato[14]:=ModBus.MB_MASTER.ReceiveBuffer.Data[4].6; (*Vedi Tabella *)
				MB_BitStato[15]:=ModBus.MB_MASTER.ReceiveBuffer.Data[4].7; (*Vedi Tabella *)
				MB_BitStato[16]:=ModBus.MB_MASTER.ReceiveBuffer.Data[5].0; (*Vedi Tabella *)
				MB_BitStato[17]:=ModBus.MB_MASTER.ReceiveBuffer.Data[5].1; (*Vedi Tabella *)
				MB_BitStato[18]:=ModBus.MB_MASTER.ReceiveBuffer.Data[5].2; (*Vedi Tabella *)
				MB_BitStato[19]:=ModBus.MB_MASTER.ReceiveBuffer.Data[5].3; (*Vedi Tabella *)
				MB_BitStato[20]:=ModBus.MB_MASTER.ReceiveBuffer.Data[5].4; (*Vedi Tabella *)
				MB_BitStato[21]:=ModBus.MB_MASTER.ReceiveBuffer.Data[5].5; (*Vedi Tabella *)
				MB_BitStato[22]:=ModBus.MB_MASTER.ReceiveBuffer.Data[5].6; (*Vedi Tabella *)
				MB_BitStato[23]:=ModBus.MB_MASTER.ReceiveBuffer.Data[5].7; (*Vedi Tabella *)
				MB_BitStato[24]:=ModBus.MB_MASTER.ReceiveBuffer.Data[6].0; (*Vedi Tabella *)
				MB_BitStato[25]:=ModBus.MB_MASTER.ReceiveBuffer.Data[6].1; (*Vedi Tabella *)
				MB_BitStato[26]:=ModBus.MB_MASTER.ReceiveBuffer.Data[6].2; (*Vedi Tabella *)
				MB_BitStato[27]:=ModBus.MB_MASTER.ReceiveBuffer.Data[6].3; (*Vedi Tabella *)
				MB_BitStato[28]:=ModBus.MB_MASTER.ReceiveBuffer.Data[6].4; (*Vedi Tabella *)
				MB_BitStato[29]:=ModBus.MB_MASTER.ReceiveBuffer.Data[6].5; (*Vedi Tabella *)
				MB_BitStato[30]:=ModBus.MB_MASTER.ReceiveBuffer.Data[6].6; (*Vedi Tabella *)
				MB_BitStato[31]:=ModBus.MB_MASTER.ReceiveBuffer.Data[6].7; (*Vedi Tabella *)
				MB_BitStato[32]:=ModBus.MB_MASTER.ReceiveBuffer.Data[7].0; (*Vedi Tabella *)
				MB_BitStato[33]:=ModBus.MB_MASTER.ReceiveBuffer.Data[7].1; (*Vedi Tabella *)
				MB_BitStato[34]:=ModBus.MB_MASTER.ReceiveBuffer.Data[7].2; (*Vedi Tabella *)
				MB_BitStato[35]:=ModBus.MB_MASTER.ReceiveBuffer.Data[7].3; (*Vedi Tabella *)
				MB_BitStato[36]:=ModBus.MB_MASTER.ReceiveBuffer.Data[7].4; (*Vedi Tabella *)
				MB_BitStato[37]:=ModBus.MB_MASTER.ReceiveBuffer.Data[7].5; (*Vedi Tabella *)
				MB_BitStato[38]:=ModBus.MB_MASTER.ReceiveBuffer.Data[7].6; (*Vedi Tabella *)
				MB_BitStato[39]:=ModBus.MB_MASTER.ReceiveBuffer.Data[7].7; (*Vedi Tabella *)
				MB_BitStato[40]:=ModBus.MB_MASTER.ReceiveBuffer.Data[8].0; (*Vedi Tabella *)
				MB_BitStato[41]:=ModBus.MB_MASTER.ReceiveBuffer.Data[8].1; (*Vedi Tabella *)
				MB_BitStato[42]:=ModBus.MB_MASTER.ReceiveBuffer.Data[8].2; (*Vedi Tabella *)
				MB_BitStato[43]:=ModBus.MB_MASTER.ReceiveBuffer.Data[8].3; (*Vedi Tabella *)
				MB_BitStato[44]:=ModBus.MB_MASTER.ReceiveBuffer.Data[8].4; (*Vedi Tabella *)
				MB_BitStato[45]:=ModBus.MB_MASTER.ReceiveBuffer.Data[8].5; (*Vedi Tabella *)
				MB_BitStato[46]:=ModBus.MB_MASTER.ReceiveBuffer.Data[8].6; (*Vedi Tabella *)
				MB_BitStato[47]:=ModBus.MB_MASTER.ReceiveBuffer.Data[8].7; (*Vedi Tabella *)
				MB_BitStato[48]:=ModBus.MB_MASTER.ReceiveBuffer.Data[9].0; (*Vedi Tabella *)
				MB_BitStato[49]:=ModBus.MB_MASTER.ReceiveBuffer.Data[9].1; (*Vedi Tabella *)
				MB_BitStato[50]:=ModBus.MB_MASTER.ReceiveBuffer.Data[9].2; (*Vedi Tabella *)
				MB_BitStato[51]:=ModBus.MB_MASTER.ReceiveBuffer.Data[9].3; (*Vedi Tabella *)
				MB_BitStato[52]:=ModBus.MB_MASTER.ReceiveBuffer.Data[9].4; (*Vedi Tabella *)
				MB_BitStato[53]:=ModBus.MB_MASTER.ReceiveBuffer.Data[9].5; (*Vedi Tabella *)
				MB_BitStato[54]:=ModBus.MB_MASTER.ReceiveBuffer.Data[9].6; (*Vedi Tabella *)
				MB_BitStato[55]:=ModBus.MB_MASTER.ReceiveBuffer.Data[9].7; (*Vedi Tabella *)
				MB_BitStato[56]:=ModBus.MB_MASTER.ReceiveBuffer.Data[10].0; (*Vedi Tabella *)
				MB_BitStato[57]:=ModBus.MB_MASTER.ReceiveBuffer.Data[10].1; (*Vedi Tabella *)
				MB_BitStato[58]:=ModBus.MB_MASTER.ReceiveBuffer.Data[10].2; (*Vedi Tabella *)
				MB_BitStato[59]:=ModBus.MB_MASTER.ReceiveBuffer.Data[10].3; (*Vedi Tabella *)
				MB_BitStato[60]:=ModBus.MB_MASTER.ReceiveBuffer.Data[10].4; (*Vedi Tabella *)
				MB_BitStato[61]:=ModBus.MB_MASTER.ReceiveBuffer.Data[10].5; (*Vedi Tabella *)
				MB_BitStato[62]:=ModBus.MB_MASTER.ReceiveBuffer.Data[10].6; (*Vedi Tabella *)
				MB_BitStato[63]:=ModBus.MB_MASTER.ReceiveBuffer.Data[10].7; (*Vedi Tabella *)

				state:=110;

			END_IF
		END_IF

	110: (* Rispota Altri paramenti *)
		IF NOT ModBus.MB_Start  THEN

			IF ModBus.MB_MASTER.MB_Error<>0 THEN
				state := 300;
			ELSE
				Modbus.MB_Query.SlaveAddress := Address;
				Modbus.MB_Query.FunctionCode := 2;
				ModBus.MB_Query.Read_StartAddress := 64;
				ModBus.MB_Query.Read_Quantity := 64;
				ModBus.MB_Start := TRUE;

				state:=115;
			END_IF
		END_IF
	115: (* Rispota Altri paramenti *)

		IF NOT ModBus.MB_Start  THEN

			IF ModBus.MB_MASTER.MB_Error<>0 THEN
				state := 300;
			ELSE

				MB_BitStato[64]:=ModBus.MB_MASTER.ReceiveBuffer.Data[3].0; (*Vedi Tabella *)
				MB_BitStato[65]:=ModBus.MB_MASTER.ReceiveBuffer.Data[3].1; (*Vedi Tabella *)
				MB_BitStato[66]:=ModBus.MB_MASTER.ReceiveBuffer.Data[3].2; (*Vedi Tabella *)
				MB_BitStato[67]:=ModBus.MB_MASTER.ReceiveBuffer.Data[3].3; (*Vedi Tabella *)
				MB_BitStato[68]:=ModBus.MB_MASTER.ReceiveBuffer.Data[3].4; (*Vedi Tabella *)
				MB_BitStato[69]:=ModBus.MB_MASTER.ReceiveBuffer.Data[3].5; (*Vedi Tabella *)
				MB_BitStato[70]:=ModBus.MB_MASTER.ReceiveBuffer.Data[3].6; (*Vedi Tabella *)
				MB_BitStato[71]:=ModBus.MB_MASTER.ReceiveBuffer.Data[3].7; (*Vedi Tabella *)
				MB_BitStato[72]:=ModBus.MB_MASTER.ReceiveBuffer.Data[4].0; (*Vedi Tabella *)
				MB_BitStato[73]:=ModBus.MB_MASTER.ReceiveBuffer.Data[4].1; (*Vedi Tabella *)
				MB_BitStato[74]:=ModBus.MB_MASTER.ReceiveBuffer.Data[4].2; (*Vedi Tabella *)
				MB_BitStato[75]:=ModBus.MB_MASTER.ReceiveBuffer.Data[4].3; (*Vedi Tabella *)
				MB_BitStato[76]:=ModBus.MB_MASTER.ReceiveBuffer.Data[4].4; (*Vedi Tabella *)
				MB_BitStato[77]:=ModBus.MB_MASTER.ReceiveBuffer.Data[4].5; (*Vedi Tabella *)
				MB_BitStato[78]:=ModBus.MB_MASTER.ReceiveBuffer.Data[4].6; (*Vedi Tabella *)
				MB_BitStato[79]:=ModBus.MB_MASTER.ReceiveBuffer.Data[4].7; (*Vedi Tabella *)
				MB_BitStato[80]:=ModBus.MB_MASTER.ReceiveBuffer.Data[5].0; (*Vedi Tabella *)
				MB_BitStato[81]:=ModBus.MB_MASTER.ReceiveBuffer.Data[5].1; (*Vedi Tabella *)
				MB_BitStato[82]:=ModBus.MB_MASTER.ReceiveBuffer.Data[5].2; (*Vedi Tabella *)
				MB_BitStato[83]:=ModBus.MB_MASTER.ReceiveBuffer.Data[5].3; (*Vedi Tabella *)
				MB_BitStato[84]:=ModBus.MB_MASTER.ReceiveBuffer.Data[5].4; (*Vedi Tabella *)
				MB_BitStato[85]:=ModBus.MB_MASTER.ReceiveBuffer.Data[5].5; (*Vedi Tabella *)
				MB_BitStato[86]:=ModBus.MB_MASTER.ReceiveBuffer.Data[5].6; (*Vedi Tabella *)
				MB_BitStato[87]:=ModBus.MB_MASTER.ReceiveBuffer.Data[5].7; (*Vedi Tabella *)
				MB_BitStato[88]:=ModBus.MB_MASTER.ReceiveBuffer.Data[6].0; (*Vedi Tabella *)
				MB_BitStato[89]:=ModBus.MB_MASTER.ReceiveBuffer.Data[6].1; (*Vedi Tabella *)
				MB_BitStato[90]:=ModBus.MB_MASTER.ReceiveBuffer.Data[6].2; (*Vedi Tabella *)
				MB_BitStato[91]:=ModBus.MB_MASTER.ReceiveBuffer.Data[6].3; (*Vedi Tabella *)
				MB_BitStato[92]:=ModBus.MB_MASTER.ReceiveBuffer.Data[6].4; (*Vedi Tabella *)
				MB_BitStato[93]:=ModBus.MB_MASTER.ReceiveBuffer.Data[6].5; (*Vedi Tabella *)
				MB_BitStato[94]:=ModBus.MB_MASTER.ReceiveBuffer.Data[6].6; (*Vedi Tabella *)
				MB_BitStato[95]:=ModBus.MB_MASTER.ReceiveBuffer.Data[6].7; (*Vedi Tabella *)
				MB_BitStato[96]:=ModBus.MB_MASTER.ReceiveBuffer.Data[7].0; (*Vedi Tabella *)
				MB_BitStato[97]:=ModBus.MB_MASTER.ReceiveBuffer.Data[7].1; (*Vedi Tabella *)
				MB_BitStato[98]:=ModBus.MB_MASTER.ReceiveBuffer.Data[7].2; (*Vedi Tabella *)
				MB_BitStato[99]:=ModBus.MB_MASTER.ReceiveBuffer.Data[7].3; (*Vedi Tabella *)
				MB_BitStato[100]:=ModBus.MB_MASTER.ReceiveBuffer.Data[7].4; (*Vedi Tabella *)
				MB_BitStato[101]:=ModBus.MB_MASTER.ReceiveBuffer.Data[7].5; (*Vedi Tabella *)
				MB_BitStato[102]:=ModBus.MB_MASTER.ReceiveBuffer.Data[7].6; (*Vedi Tabella *)
				MB_BitStato[103]:=ModBus.MB_MASTER.ReceiveBuffer.Data[7].7; (*Vedi Tabella *)
				MB_BitStato[104]:=ModBus.MB_MASTER.ReceiveBuffer.Data[8].0; (*Vedi Tabella *)
				MB_BitStato[105]:=ModBus.MB_MASTER.ReceiveBuffer.Data[8].1; (*Vedi Tabella *)
				MB_BitStato[106]:=ModBus.MB_MASTER.ReceiveBuffer.Data[8].2; (*Vedi Tabella *)
				MB_BitStato[107]:=ModBus.MB_MASTER.ReceiveBuffer.Data[8].3; (*Vedi Tabella *)
				MB_BitStato[108]:=ModBus.MB_MASTER.ReceiveBuffer.Data[8].4; (*Vedi Tabella *)
				MB_BitStato[109]:=ModBus.MB_MASTER.ReceiveBuffer.Data[8].5; (*Vedi Tabella *)
				MB_BitStato[110]:=ModBus.MB_MASTER.ReceiveBuffer.Data[8].6; (*Vedi Tabella *)
				MB_BitStato[111]:=ModBus.MB_MASTER.ReceiveBuffer.Data[8].7; (*Vedi Tabella *)
				MB_BitStato[112]:=ModBus.MB_MASTER.ReceiveBuffer.Data[9].0; (*Vedi Tabella *)
				MB_BitStato[113]:=ModBus.MB_MASTER.ReceiveBuffer.Data[9].1; (*Vedi Tabella *)
				MB_BitStato[114]:=ModBus.MB_MASTER.ReceiveBuffer.Data[9].2; (*Vedi Tabella *)
				MB_BitStato[115]:=ModBus.MB_MASTER.ReceiveBuffer.Data[9].3; (*Vedi Tabella *)
				MB_BitStato[116]:=ModBus.MB_MASTER.ReceiveBuffer.Data[9].4; (*Vedi Tabella *)
				MB_BitStato[117]:=ModBus.MB_MASTER.ReceiveBuffer.Data[9].5; (*Vedi Tabella *)
				MB_BitStato[118]:=ModBus.MB_MASTER.ReceiveBuffer.Data[9].6; (*Vedi Tabella *)
				MB_BitStato[119]:=ModBus.MB_MASTER.ReceiveBuffer.Data[9].7; (*Vedi Tabella *)
				MB_BitStato[120]:=ModBus.MB_MASTER.ReceiveBuffer.Data[10].0; (*Vedi Tabella *)
				MB_BitStato[121]:=ModBus.MB_MASTER.ReceiveBuffer.Data[10].1; (*Vedi Tabella *)
				MB_BitStato[122]:=ModBus.MB_MASTER.ReceiveBuffer.Data[10].2; (*Vedi Tabella *)
				MB_BitStato[123]:=ModBus.MB_MASTER.ReceiveBuffer.Data[10].3; (*Vedi Tabella *)
				MB_BitStato[124]:=ModBus.MB_MASTER.ReceiveBuffer.Data[10].4; (*Vedi Tabella *)
				MB_BitStato[125]:=ModBus.MB_MASTER.ReceiveBuffer.Data[10].5; (*Vedi Tabella *)
				MB_BitStato[126]:=ModBus.MB_MASTER.ReceiveBuffer.Data[10].6; (*Vedi Tabella *)
				MB_BitStato[127]:=ModBus.MB_MASTER.ReceiveBuffer.Data[10].7; (*Vedi Tabella *)


				state:=120;

			END_IF
		END_IF


	120: (* Rispota Altri paramenti *)
		IF NOT ModBus.MB_Start  THEN

			IF ModBus.MB_MASTER.MB_Error<>0 THEN
				state := 300;
			ELSE
				Modbus.MB_Query.SlaveAddress := Address;
				Modbus.MB_Query.FunctionCode := 2;
				ModBus.MB_Query.Read_StartAddress := 128;
				ModBus.MB_Query.Read_Quantity := 64;
				ModBus.MB_Start := TRUE;

				state:=125;
			END_IF
		END_IF
	125: (* Rispota Altri paramenti *)

		IF NOT ModBus.MB_Start  THEN

			IF ModBus.MB_MASTER.MB_Error<>0 THEN
				state := 300;
			ELSE

				MB_BitStato[128]:=ModBus.MB_MASTER.ReceiveBuffer.Data[3].0; (*Vedi Tabella *)
				MB_BitStato[129]:=ModBus.MB_MASTER.ReceiveBuffer.Data[3].1; (*Vedi Tabella *)
				MB_BitStato[130]:=ModBus.MB_MASTER.ReceiveBuffer.Data[3].2; (*Vedi Tabella *)
				MB_BitStato[131]:=ModBus.MB_MASTER.ReceiveBuffer.Data[3].3; (*Vedi Tabella *)
				MB_BitStato[132]:=ModBus.MB_MASTER.ReceiveBuffer.Data[3].4; (*Vedi Tabella *)
				MB_BitStato[133]:=ModBus.MB_MASTER.ReceiveBuffer.Data[3].5; (*Vedi Tabella *)
				MB_BitStato[134]:=ModBus.MB_MASTER.ReceiveBuffer.Data[3].6; (*Vedi Tabella *)
				MB_BitStato[135]:=ModBus.MB_MASTER.ReceiveBuffer.Data[3].7; (*Vedi Tabella *)
				MB_BitStato[136]:=ModBus.MB_MASTER.ReceiveBuffer.Data[4].0; (*Vedi Tabella *)
				MB_BitStato[137]:=ModBus.MB_MASTER.ReceiveBuffer.Data[4].1; (*Vedi Tabella *)
				MB_BitStato[138]:=ModBus.MB_MASTER.ReceiveBuffer.Data[4].2; (*Vedi Tabella *)
				MB_BitStato[139]:=ModBus.MB_MASTER.ReceiveBuffer.Data[4].3; (*Vedi Tabella *)
				MB_BitStato[140]:=ModBus.MB_MASTER.ReceiveBuffer.Data[4].4; (*Vedi Tabella *)
				MB_BitStato[141]:=ModBus.MB_MASTER.ReceiveBuffer.Data[4].5; (*Vedi Tabella *)
				MB_BitStato[142]:=ModBus.MB_MASTER.ReceiveBuffer.Data[4].6; (*Vedi Tabella *)
				MB_BitStato[143]:=ModBus.MB_MASTER.ReceiveBuffer.Data[4].7; (*Vedi Tabella *)
				MB_BitStato[144]:=ModBus.MB_MASTER.ReceiveBuffer.Data[5].0; (*Vedi Tabella *)
				MB_BitStato[145]:=ModBus.MB_MASTER.ReceiveBuffer.Data[5].1; (*Vedi Tabella *)
				MB_BitStato[146]:=ModBus.MB_MASTER.ReceiveBuffer.Data[5].2; (*Vedi Tabella *)
				MB_BitStato[147]:=ModBus.MB_MASTER.ReceiveBuffer.Data[5].3; (*Vedi Tabella *)
				MB_BitStato[148]:=ModBus.MB_MASTER.ReceiveBuffer.Data[5].4; (*Vedi Tabella *)
				MB_BitStato[149]:=ModBus.MB_MASTER.ReceiveBuffer.Data[5].5; (*Vedi Tabella *)
				MB_BitStato[150]:=ModBus.MB_MASTER.ReceiveBuffer.Data[5].6; (*Vedi Tabella *)
				MB_BitStato[151]:=ModBus.MB_MASTER.ReceiveBuffer.Data[5].7; (*Vedi Tabella *)
				MB_BitStato[152]:=ModBus.MB_MASTER.ReceiveBuffer.Data[6].0; (*Vedi Tabella *)
				MB_BitStato[153]:=ModBus.MB_MASTER.ReceiveBuffer.Data[6].1; (*Vedi Tabella *)
				MB_BitStato[154]:=ModBus.MB_MASTER.ReceiveBuffer.Data[6].2; (*Vedi Tabella *)
				MB_BitStato[155]:=ModBus.MB_MASTER.ReceiveBuffer.Data[6].3; (*Vedi Tabella *)
				MB_BitStato[156]:=ModBus.MB_MASTER.ReceiveBuffer.Data[6].4; (*Vedi Tabella *)
				MB_BitStato[157]:=ModBus.MB_MASTER.ReceiveBuffer.Data[6].5; (*Vedi Tabella *)
				MB_BitStato[158]:=ModBus.MB_MASTER.ReceiveBuffer.Data[6].6; (*Vedi Tabella *)
				MB_BitStato[159]:=ModBus.MB_MASTER.ReceiveBuffer.Data[6].7; (*Vedi Tabella *)
				MB_BitStato[160]:=ModBus.MB_MASTER.ReceiveBuffer.Data[7].0; (*Vedi Tabella *)
				MB_BitStato[161]:=ModBus.MB_MASTER.ReceiveBuffer.Data[7].1; (*Vedi Tabella *)
				MB_BitStato[162]:=ModBus.MB_MASTER.ReceiveBuffer.Data[7].2; (*Vedi Tabella *)
				MB_BitStato[163]:=ModBus.MB_MASTER.ReceiveBuffer.Data[7].3; (*Vedi Tabella *)
				MB_BitStato[164]:=ModBus.MB_MASTER.ReceiveBuffer.Data[7].4; (*Vedi Tabella *)
				MB_BitStato[165]:=ModBus.MB_MASTER.ReceiveBuffer.Data[7].5; (*Vedi Tabella *)
				MB_BitStato[166]:=ModBus.MB_MASTER.ReceiveBuffer.Data[7].6; (*Vedi Tabella *)
				MB_BitStato[167]:=ModBus.MB_MASTER.ReceiveBuffer.Data[7].7; (*Vedi Tabella *)
				MB_BitStato[168]:=ModBus.MB_MASTER.ReceiveBuffer.Data[8].0; (*Vedi Tabella *)
				MB_BitStato[169]:=ModBus.MB_MASTER.ReceiveBuffer.Data[8].1; (*Vedi Tabella *)
				MB_BitStato[170]:=ModBus.MB_MASTER.ReceiveBuffer.Data[8].2; (*Vedi Tabella *)
				MB_BitStato[171]:=ModBus.MB_MASTER.ReceiveBuffer.Data[8].3; (*Vedi Tabella *)
				MB_BitStato[172]:=ModBus.MB_MASTER.ReceiveBuffer.Data[8].4; (*Vedi Tabella *)
				MB_BitStato[173]:=ModBus.MB_MASTER.ReceiveBuffer.Data[8].5; (*Vedi Tabella *)
				MB_BitStato[174]:=ModBus.MB_MASTER.ReceiveBuffer.Data[8].6; (*Vedi Tabella *)
				MB_BitStato[175]:=ModBus.MB_MASTER.ReceiveBuffer.Data[8].7; (*Vedi Tabella *)
				MB_BitStato[176]:=ModBus.MB_MASTER.ReceiveBuffer.Data[9].0; (*Vedi Tabella *)
				MB_BitStato[177]:=ModBus.MB_MASTER.ReceiveBuffer.Data[9].1; (*Vedi Tabella *)
				MB_BitStato[178]:=ModBus.MB_MASTER.ReceiveBuffer.Data[9].2; (*Vedi Tabella *)
				MB_BitStato[179]:=ModBus.MB_MASTER.ReceiveBuffer.Data[9].3; (*Vedi Tabella *)
				MB_BitStato[180]:=ModBus.MB_MASTER.ReceiveBuffer.Data[9].4; (*Vedi Tabella *)
				MB_BitStato[181]:=ModBus.MB_MASTER.ReceiveBuffer.Data[9].5; (*Vedi Tabella *)
				MB_BitStato[182]:=ModBus.MB_MASTER.ReceiveBuffer.Data[9].6; (*Vedi Tabella *)
				MB_BitStato[183]:=ModBus.MB_MASTER.ReceiveBuffer.Data[9].7; (*Vedi Tabella *)
				MB_BitStato[184]:=ModBus.MB_MASTER.ReceiveBuffer.Data[10].0; (*Vedi Tabella *)
				MB_BitStato[185]:=ModBus.MB_MASTER.ReceiveBuffer.Data[10].1; (*Vedi Tabella *)
				MB_BitStato[186]:=ModBus.MB_MASTER.ReceiveBuffer.Data[10].2; (*Vedi Tabella *)
				MB_BitStato[187]:=ModBus.MB_MASTER.ReceiveBuffer.Data[10].3; (*Vedi Tabella *)
				MB_BitStato[188]:=ModBus.MB_MASTER.ReceiveBuffer.Data[10].4; (*Vedi Tabella *)
				MB_BitStato[189]:=ModBus.MB_MASTER.ReceiveBuffer.Data[10].5; (*Vedi Tabella *)
				MB_BitStato[190]:=ModBus.MB_MASTER.ReceiveBuffer.Data[10].6; (*Vedi Tabella *)
				MB_BitStato[191]:=ModBus.MB_MASTER.ReceiveBuffer.Data[10].7; (*Vedi Tabella *)


				state:=130;

			END_IF
		END_IF


	130: (* Rispota Altri paramenti COIL *)
		IF NOT ModBus.MB_Start  THEN

			IF ModBus.MB_MASTER.MB_Error<>0 THEN
				state := 300;
			ELSE
				Modbus.MB_Query.SlaveAddress := Address;
				Modbus.MB_Query.FunctionCode := 2;
				ModBus.MB_Query.Read_StartAddress := 192;	(* richiedo lettura altri Parametri *)
				ModBus.MB_Query.Read_Quantity := 64;
				ModBus.MB_Start := TRUE;

				state:=135;
			END_IF
		END_IF
	135: (* Rispota Altri paramenti *)

		IF NOT ModBus.MB_Start  THEN

			IF ModBus.MB_MASTER.MB_Error<>0 THEN
				state := 300;
			ELSE

				MB_BitStato[192]:=ModBus.MB_MASTER.ReceiveBuffer.Data[3].0; (*Vedi Tabella *)
				MB_BitStato[193]:=ModBus.MB_MASTER.ReceiveBuffer.Data[3].1; (*Vedi Tabella *)
				MB_BitStato[194]:=ModBus.MB_MASTER.ReceiveBuffer.Data[3].2; (*Vedi Tabella *)
				MB_BitStato[195]:=ModBus.MB_MASTER.ReceiveBuffer.Data[3].3; (*Vedi Tabella *)
				MB_BitStato[196]:=ModBus.MB_MASTER.ReceiveBuffer.Data[3].4; (*Vedi Tabella *)
				MB_BitStato[197]:=ModBus.MB_MASTER.ReceiveBuffer.Data[3].5; (*Vedi Tabella *)
				MB_BitStato[198]:=ModBus.MB_MASTER.ReceiveBuffer.Data[3].6; (*Vedi Tabella *)
				MB_BitStato[199]:=ModBus.MB_MASTER.ReceiveBuffer.Data[3].7; (*Vedi Tabella *)
				MB_BitStato[200]:=ModBus.MB_MASTER.ReceiveBuffer.Data[4].0; (*Vedi Tabella *)
				MB_BitStato[201]:=ModBus.MB_MASTER.ReceiveBuffer.Data[4].1; (*Vedi Tabella *)
				MB_BitStato[202]:=ModBus.MB_MASTER.ReceiveBuffer.Data[4].2; (*Vedi Tabella *)
				MB_BitStato[203]:=ModBus.MB_MASTER.ReceiveBuffer.Data[4].3; (*Vedi Tabella *)
				MB_BitStato[204]:=ModBus.MB_MASTER.ReceiveBuffer.Data[4].4; (*Vedi Tabella *)
				MB_BitStato[205]:=ModBus.MB_MASTER.ReceiveBuffer.Data[4].5; (*Vedi Tabella *)
				MB_BitStato[206]:=ModBus.MB_MASTER.ReceiveBuffer.Data[4].6; (*Vedi Tabella *)
				MB_BitStato[207]:=ModBus.MB_MASTER.ReceiveBuffer.Data[4].7; (*Vedi Tabella *)
				MB_BitStato[208]:=ModBus.MB_MASTER.ReceiveBuffer.Data[5].0; (*Vedi Tabella *)
				MB_BitStato[209]:=ModBus.MB_MASTER.ReceiveBuffer.Data[5].1; (*Vedi Tabella *)
				MB_BitStato[210]:=ModBus.MB_MASTER.ReceiveBuffer.Data[5].2; (*Vedi Tabella *)
				MB_BitStato[211]:=ModBus.MB_MASTER.ReceiveBuffer.Data[5].3; (*Vedi Tabella *)
				MB_BitStato[212]:=ModBus.MB_MASTER.ReceiveBuffer.Data[5].4; (*Vedi Tabella *)
				MB_BitStato[213]:=ModBus.MB_MASTER.ReceiveBuffer.Data[5].5; (*Vedi Tabella *)
				MB_BitStato[214]:=ModBus.MB_MASTER.ReceiveBuffer.Data[5].6; (*Vedi Tabella *)
				MB_BitStato[215]:=ModBus.MB_MASTER.ReceiveBuffer.Data[5].7; (*Vedi Tabella *)
				MB_BitStato[216]:=ModBus.MB_MASTER.ReceiveBuffer.Data[6].0; (*Vedi Tabella *)
				MB_BitStato[217]:=ModBus.MB_MASTER.ReceiveBuffer.Data[6].1; (*Vedi Tabella *)
				MB_BitStato[218]:=ModBus.MB_MASTER.ReceiveBuffer.Data[6].2; (*Vedi Tabella *)
				MB_BitStato[219]:=ModBus.MB_MASTER.ReceiveBuffer.Data[6].3; (*Vedi Tabella *)
				MB_BitStato[220]:=ModBus.MB_MASTER.ReceiveBuffer.Data[6].4; (*Vedi Tabella *)
				MB_BitStato[221]:=ModBus.MB_MASTER.ReceiveBuffer.Data[6].5; (*Vedi Tabella *)
				MB_BitStato[222]:=ModBus.MB_MASTER.ReceiveBuffer.Data[6].6; (*Vedi Tabella *)
				MB_BitStato[223]:=ModBus.MB_MASTER.ReceiveBuffer.Data[6].7; (*Vedi Tabella *)
				MB_BitStato[224]:=ModBus.MB_MASTER.ReceiveBuffer.Data[7].0; (*Vedi Tabella *)
				MB_BitStato[225]:=ModBus.MB_MASTER.ReceiveBuffer.Data[7].1; (*Vedi Tabella *)
				MB_BitStato[226]:=ModBus.MB_MASTER.ReceiveBuffer.Data[7].2; (*Vedi Tabella *)
				MB_BitStato[227]:=ModBus.MB_MASTER.ReceiveBuffer.Data[7].3; (*Vedi Tabella *)
				MB_BitStato[228]:=ModBus.MB_MASTER.ReceiveBuffer.Data[7].4; (*Vedi Tabella *)
				MB_BitStato[229]:=ModBus.MB_MASTER.ReceiveBuffer.Data[7].5; (*Vedi Tabella *)
				MB_BitStato[230]:=ModBus.MB_MASTER.ReceiveBuffer.Data[7].6; (*Vedi Tabella *)
				MB_BitStato[231]:=ModBus.MB_MASTER.ReceiveBuffer.Data[7].7; (*Vedi Tabella *)
				MB_BitStato[232]:=ModBus.MB_MASTER.ReceiveBuffer.Data[8].0; (*Vedi Tabella *)
				MB_BitStato[233]:=ModBus.MB_MASTER.ReceiveBuffer.Data[8].1; (*Vedi Tabella *)
				MB_BitStato[234]:=ModBus.MB_MASTER.ReceiveBuffer.Data[8].2; (*Vedi Tabella *)
				MB_BitStato[235]:=ModBus.MB_MASTER.ReceiveBuffer.Data[8].3; (*Vedi Tabella *)
				MB_BitStato[236]:=ModBus.MB_MASTER.ReceiveBuffer.Data[8].4; (*Vedi Tabella *)
				MB_BitStato[237]:=ModBus.MB_MASTER.ReceiveBuffer.Data[8].5; (*Vedi Tabella *)
				MB_BitStato[238]:=ModBus.MB_MASTER.ReceiveBuffer.Data[8].6; (*Vedi Tabella *)
				MB_BitStato[239]:=ModBus.MB_MASTER.ReceiveBuffer.Data[8].7; (*Vedi Tabella *)
				MB_BitStato[240]:=ModBus.MB_MASTER.ReceiveBuffer.Data[9].0; (*Vedi Tabella *)
				MB_BitStato[241]:=ModBus.MB_MASTER.ReceiveBuffer.Data[9].1; (*Vedi Tabella *)
				MB_BitStato[242]:=ModBus.MB_MASTER.ReceiveBuffer.Data[9].2; (*Vedi Tabella *)
				MB_BitStato[243]:=ModBus.MB_MASTER.ReceiveBuffer.Data[9].3; (*Vedi Tabella *)
				MB_BitStato[244]:=ModBus.MB_MASTER.ReceiveBuffer.Data[9].4; (*Vedi Tabella *)
				MB_BitStato[245]:=ModBus.MB_MASTER.ReceiveBuffer.Data[9].5; (*Vedi Tabella *)
				MB_BitStato[246]:=ModBus.MB_MASTER.ReceiveBuffer.Data[9].6; (*Vedi Tabella *)
				MB_BitStato[247]:=ModBus.MB_MASTER.ReceiveBuffer.Data[9].7; (*Vedi Tabella *)
				MB_BitStato[248]:=ModBus.MB_MASTER.ReceiveBuffer.Data[10].0; (*Vedi Tabella *)
				MB_BitStato[249]:=ModBus.MB_MASTER.ReceiveBuffer.Data[10].1; (*Vedi Tabella *)
				MB_BitStato[250]:=ModBus.MB_MASTER.ReceiveBuffer.Data[10].2; (*Vedi Tabella *)
				MB_BitStato[251]:=ModBus.MB_MASTER.ReceiveBuffer.Data[10].3; (*Vedi Tabella *)
				MB_BitStato[252]:=ModBus.MB_MASTER.ReceiveBuffer.Data[10].4; (*Vedi Tabella *)
				MB_BitStato[253]:=ModBus.MB_MASTER.ReceiveBuffer.Data[10].5; (*Vedi Tabella *)
				MB_BitStato[254]:=ModBus.MB_MASTER.ReceiveBuffer.Data[10].6; (*Vedi Tabella *)
				MB_BitStato[255]:=ModBus.MB_MASTER.ReceiveBuffer.Data[10].7; (*Vedi Tabella *)

				state:=140;

			END_IF
		END_IF

	140: (* Rispota Altri paramenti COIL *)
		IF NOT ModBus.MB_Start  THEN

			IF ModBus.MB_MASTER.MB_Error<>0 THEN
				state := 300;
			ELSE
				Modbus.MB_Query.SlaveAddress := Address;
				Modbus.MB_Query.FunctionCode := 2;
				ModBus.MB_Query.Read_StartAddress := 256;	(* richiedo lettura altri Parametri *)
				ModBus.MB_Query.Read_Quantity := 64;
				ModBus.MB_Start := TRUE;

				state:=145;
			END_IF
		END_IF
	145: (* Rispota Altri paramenti *)

		IF NOT ModBus.MB_Start  THEN

			IF ModBus.MB_MASTER.MB_Error<>0 THEN
				state := 300;
			ELSE

				MB_BitStato[256]:=ModBus.MB_MASTER.ReceiveBuffer.Data[3].0; (*Vedi Tabella *)
				MB_BitStato[257]:=ModBus.MB_MASTER.ReceiveBuffer.Data[3].1; (*Vedi Tabella *)
				MB_BitStato[258]:=ModBus.MB_MASTER.ReceiveBuffer.Data[3].2; (*Vedi Tabella *)
				MB_BitStato[259]:=ModBus.MB_MASTER.ReceiveBuffer.Data[3].3; (*Vedi Tabella *)
				MB_BitStato[260]:=ModBus.MB_MASTER.ReceiveBuffer.Data[3].4; (*Vedi Tabella *)
				MB_BitStato[261]:=ModBus.MB_MASTER.ReceiveBuffer.Data[3].5; (*Vedi Tabella *)
				MB_BitStato[262]:=ModBus.MB_MASTER.ReceiveBuffer.Data[3].6; (*Vedi Tabella *)
				MB_BitStato[263]:=ModBus.MB_MASTER.ReceiveBuffer.Data[3].7; (*Vedi Tabella *)
				MB_BitStato[264]:=ModBus.MB_MASTER.ReceiveBuffer.Data[4].0; (*Vedi Tabella *)
				MB_BitStato[265]:=ModBus.MB_MASTER.ReceiveBuffer.Data[4].1; (*Vedi Tabella *)
				MB_BitStato[266]:=ModBus.MB_MASTER.ReceiveBuffer.Data[4].2; (*Vedi Tabella *)
				MB_BitStato[267]:=ModBus.MB_MASTER.ReceiveBuffer.Data[4].3; (*Vedi Tabella *)
				MB_BitStato[268]:=ModBus.MB_MASTER.ReceiveBuffer.Data[4].4; (*Vedi Tabella *)
				MB_BitStato[269]:=ModBus.MB_MASTER.ReceiveBuffer.Data[4].5; (*Vedi Tabella *)
				MB_BitStato[270]:=ModBus.MB_MASTER.ReceiveBuffer.Data[4].6; (*Vedi Tabella *)
				MB_BitStato[271]:=ModBus.MB_MASTER.ReceiveBuffer.Data[4].7; (*Vedi Tabella *)
				MB_BitStato[272]:=ModBus.MB_MASTER.ReceiveBuffer.Data[5].0; (*Vedi Tabella *)
				MB_BitStato[273]:=ModBus.MB_MASTER.ReceiveBuffer.Data[5].1; (*Vedi Tabella *)
				MB_BitStato[274]:=ModBus.MB_MASTER.ReceiveBuffer.Data[5].2; (*Vedi Tabella *)
				MB_BitStato[275]:=ModBus.MB_MASTER.ReceiveBuffer.Data[5].3; (*Vedi Tabella *)
				MB_BitStato[276]:=ModBus.MB_MASTER.ReceiveBuffer.Data[5].4; (*Vedi Tabella *)
				MB_BitStato[277]:=ModBus.MB_MASTER.ReceiveBuffer.Data[5].5; (*Vedi Tabella *)
				MB_BitStato[278]:=ModBus.MB_MASTER.ReceiveBuffer.Data[5].6; (*Vedi Tabella *)
				MB_BitStato[279]:=ModBus.MB_MASTER.ReceiveBuffer.Data[5].7; (*Vedi Tabella *)
				MB_BitStato[280]:=ModBus.MB_MASTER.ReceiveBuffer.Data[6].0; (*Vedi Tabella *)
				MB_BitStato[281]:=ModBus.MB_MASTER.ReceiveBuffer.Data[6].1; (*Vedi Tabella *)
				MB_BitStato[282]:=ModBus.MB_MASTER.ReceiveBuffer.Data[6].2; (*Vedi Tabella *)
				MB_BitStato[283]:=ModBus.MB_MASTER.ReceiveBuffer.Data[6].3; (*Vedi Tabella *)
				MB_BitStato[284]:=ModBus.MB_MASTER.ReceiveBuffer.Data[6].4; (*Vedi Tabella *)
				MB_BitStato[285]:=ModBus.MB_MASTER.ReceiveBuffer.Data[6].5; (*Vedi Tabella *)
				MB_BitStato[286]:=ModBus.MB_MASTER.ReceiveBuffer.Data[6].6; (*Vedi Tabella *)
				MB_BitStato[287]:=ModBus.MB_MASTER.ReceiveBuffer.Data[6].7; (*Vedi Tabella *)
				MB_BitStato[288]:=ModBus.MB_MASTER.ReceiveBuffer.Data[7].0; (*Vedi Tabella *)
				MB_BitStato[289]:=ModBus.MB_MASTER.ReceiveBuffer.Data[7].1; (*Vedi Tabella *)
				MB_BitStato[290]:=ModBus.MB_MASTER.ReceiveBuffer.Data[7].2; (*Vedi Tabella *)
				MB_BitStato[291]:=ModBus.MB_MASTER.ReceiveBuffer.Data[7].3; (*Vedi Tabella *)
				MB_BitStato[292]:=ModBus.MB_MASTER.ReceiveBuffer.Data[7].4; (*Vedi Tabella *)
				MB_BitStato[293]:=ModBus.MB_MASTER.ReceiveBuffer.Data[7].5; (*Vedi Tabella *)
				MB_BitStato[294]:=ModBus.MB_MASTER.ReceiveBuffer.Data[7].6; (*Vedi Tabella *)
				MB_BitStato[295]:=ModBus.MB_MASTER.ReceiveBuffer.Data[7].7; (*Vedi Tabella *)
				MB_BitStato[296]:=ModBus.MB_MASTER.ReceiveBuffer.Data[8].0; (*Vedi Tabella *)
				MB_BitStato[297]:=ModBus.MB_MASTER.ReceiveBuffer.Data[8].1; (*Vedi Tabella *)
				MB_BitStato[298]:=ModBus.MB_MASTER.ReceiveBuffer.Data[8].2; (*Vedi Tabella *)
				MB_BitStato[299]:=ModBus.MB_MASTER.ReceiveBuffer.Data[8].3; (*Vedi Tabella *)
				MB_BitStato[300]:=ModBus.MB_MASTER.ReceiveBuffer.Data[8].4; (*Vedi Tabella *)
				MB_BitStato[301]:=ModBus.MB_MASTER.ReceiveBuffer.Data[8].5; (*Vedi Tabella *)
				MB_BitStato[302]:=ModBus.MB_MASTER.ReceiveBuffer.Data[8].6; (*Vedi Tabella *)
				MB_BitStato[303]:=ModBus.MB_MASTER.ReceiveBuffer.Data[8].7; (*Vedi Tabella *)
				MB_BitStato[304]:=ModBus.MB_MASTER.ReceiveBuffer.Data[9].0; (*Vedi Tabella *)
				MB_BitStato[305]:=ModBus.MB_MASTER.ReceiveBuffer.Data[9].1; (*Vedi Tabella *)
				MB_BitStato[306]:=ModBus.MB_MASTER.ReceiveBuffer.Data[9].2; (*Vedi Tabella *)
				MB_BitStato[307]:=ModBus.MB_MASTER.ReceiveBuffer.Data[9].3; (*Vedi Tabella *)
				MB_BitStato[308]:=ModBus.MB_MASTER.ReceiveBuffer.Data[9].4; (*Vedi Tabella *)
				MB_BitStato[309]:=ModBus.MB_MASTER.ReceiveBuffer.Data[9].5; (*Vedi Tabella *)
				MB_BitStato[310]:=ModBus.MB_MASTER.ReceiveBuffer.Data[9].6; (*Vedi Tabella *)
				MB_BitStato[311]:=ModBus.MB_MASTER.ReceiveBuffer.Data[9].7; (*Vedi Tabella *)
				MB_BitStato[312]:=ModBus.MB_MASTER.ReceiveBuffer.Data[10].0; (*Vedi Tabella *)
				MB_BitStato[313]:=ModBus.MB_MASTER.ReceiveBuffer.Data[10].1; (*Vedi Tabella *)
				MB_BitStato[314]:=ModBus.MB_MASTER.ReceiveBuffer.Data[10].2; (*Vedi Tabella *)
				MB_BitStato[315]:=ModBus.MB_MASTER.ReceiveBuffer.Data[10].3; (*Vedi Tabella *)
				MB_BitStato[316]:=ModBus.MB_MASTER.ReceiveBuffer.Data[10].4; (*Vedi Tabella *)
				MB_BitStato[317]:=ModBus.MB_MASTER.ReceiveBuffer.Data[10].5; (*Vedi Tabella *)
				MB_BitStato[318]:=ModBus.MB_MASTER.ReceiveBuffer.Data[10].6; (*Vedi Tabella *)
				MB_BitStato[319]:=ModBus.MB_MASTER.ReceiveBuffer.Data[10].7; (*Vedi Tabella *)

				state:=160;

			END_IF
		END_IF

	160: (* Rispota Altri paramenti COIL *)
		IF NOT ModBus.MB_Start  THEN

			IF ModBus.MB_MASTER.MB_Error<>0 THEN
				state := 300;
			ELSE
				Modbus.MB_Query.SlaveAddress := Address;
				Modbus.MB_Query.FunctionCode := 2;
				ModBus.MB_Query.Read_StartAddress := 320;	(* richiedo lettura altri Parametri *)
				ModBus.MB_Query.Read_Quantity := 64;
				ModBus.MB_Start := TRUE;

				state:=165;
			END_IF
		END_IF
	165: (* Rispota Altri paramenti *)

		IF NOT ModBus.MB_Start  THEN

			IF ModBus.MB_MASTER.MB_Error<>0 THEN
				state := 300;
			ELSE

				MB_BitStato[320]:=ModBus.MB_MASTER.ReceiveBuffer.Data[3].0; (*Vedi Tabella *)
				MB_BitStato[321]:=ModBus.MB_MASTER.ReceiveBuffer.Data[3].1; (*Vedi Tabella *)
				MB_BitStato[322]:=ModBus.MB_MASTER.ReceiveBuffer.Data[3].2; (*Vedi Tabella *)
				MB_BitStato[323]:=ModBus.MB_MASTER.ReceiveBuffer.Data[3].3; (*Vedi Tabella *)
				MB_BitStato[324]:=ModBus.MB_MASTER.ReceiveBuffer.Data[3].4; (*Vedi Tabella *)
				MB_BitStato[325]:=ModBus.MB_MASTER.ReceiveBuffer.Data[3].5; (*Vedi Tabella *)
				MB_BitStato[326]:=ModBus.MB_MASTER.ReceiveBuffer.Data[3].6; (*Vedi Tabella *)
				MB_BitStato[327]:=ModBus.MB_MASTER.ReceiveBuffer.Data[3].7; (*Vedi Tabella *)
				MB_BitStato[328]:=ModBus.MB_MASTER.ReceiveBuffer.Data[4].0; (*Vedi Tabella *)
				MB_BitStato[329]:=ModBus.MB_MASTER.ReceiveBuffer.Data[4].1; (*Vedi Tabella *)
				MB_BitStato[330]:=ModBus.MB_MASTER.ReceiveBuffer.Data[4].2; (*Vedi Tabella *)
				MB_BitStato[331]:=ModBus.MB_MASTER.ReceiveBuffer.Data[4].3; (*Vedi Tabella *)
				MB_BitStato[332]:=ModBus.MB_MASTER.ReceiveBuffer.Data[4].4; (*Vedi Tabella *)
				MB_BitStato[333]:=ModBus.MB_MASTER.ReceiveBuffer.Data[4].5; (*Vedi Tabella *)
				MB_BitStato[334]:=ModBus.MB_MASTER.ReceiveBuffer.Data[4].6; (*Vedi Tabella *)
				MB_BitStato[335]:=ModBus.MB_MASTER.ReceiveBuffer.Data[4].7; (*Vedi Tabella *)
				MB_BitStato[336]:=ModBus.MB_MASTER.ReceiveBuffer.Data[5].0; (*Vedi Tabella *)
				MB_BitStato[337]:=ModBus.MB_MASTER.ReceiveBuffer.Data[5].1; (*Vedi Tabella *)
				MB_BitStato[338]:=ModBus.MB_MASTER.ReceiveBuffer.Data[5].2; (*Vedi Tabella *)
				MB_BitStato[339]:=ModBus.MB_MASTER.ReceiveBuffer.Data[5].3; (*Vedi Tabella *)
				MB_BitStato[340]:=ModBus.MB_MASTER.ReceiveBuffer.Data[5].4; (*Vedi Tabella *)
				MB_BitStato[341]:=ModBus.MB_MASTER.ReceiveBuffer.Data[5].5; (*Vedi Tabella *)
				MB_BitStato[342]:=ModBus.MB_MASTER.ReceiveBuffer.Data[5].6; (*Vedi Tabella *)
				MB_BitStato[343]:=ModBus.MB_MASTER.ReceiveBuffer.Data[5].7; (*Vedi Tabella *)
				MB_BitStato[344]:=ModBus.MB_MASTER.ReceiveBuffer.Data[6].0; (*Vedi Tabella *)
				MB_BitStato[345]:=ModBus.MB_MASTER.ReceiveBuffer.Data[6].1; (*Vedi Tabella *)
				MB_BitStato[346]:=ModBus.MB_MASTER.ReceiveBuffer.Data[6].2; (*Vedi Tabella *)
				MB_BitStato[347]:=ModBus.MB_MASTER.ReceiveBuffer.Data[6].3; (*Vedi Tabella *)
				MB_BitStato[348]:=ModBus.MB_MASTER.ReceiveBuffer.Data[6].4; (*Vedi Tabella *)
				MB_BitStato[349]:=ModBus.MB_MASTER.ReceiveBuffer.Data[6].5; (*Vedi Tabella *)
				MB_BitStato[350]:=ModBus.MB_MASTER.ReceiveBuffer.Data[6].6; (*Vedi Tabella *)
				MB_BitStato[351]:=ModBus.MB_MASTER.ReceiveBuffer.Data[6].7; (*Vedi Tabella *)
				MB_BitStato[352]:=ModBus.MB_MASTER.ReceiveBuffer.Data[7].0; (*Vedi Tabella *)
				MB_BitStato[353]:=ModBus.MB_MASTER.ReceiveBuffer.Data[7].1; (*Vedi Tabella *)
				MB_BitStato[354]:=ModBus.MB_MASTER.ReceiveBuffer.Data[7].2; (*Vedi Tabella *)
				MB_BitStato[355]:=ModBus.MB_MASTER.ReceiveBuffer.Data[7].3; (*Vedi Tabella *)
				MB_BitStato[356]:=ModBus.MB_MASTER.ReceiveBuffer.Data[7].4; (*Vedi Tabella *)
				MB_BitStato[357]:=ModBus.MB_MASTER.ReceiveBuffer.Data[7].5; (*Vedi Tabella *)
	(*			MB_BitStato[359]:=ModBus.MB_MASTER.ReceiveBuffer.Data[7].6; (*Vedi Tabella *)
				MB_BitStato[360]:=ModBus.MB_MASTER.ReceiveBuffer.Data[7].7; (*Vedi Tabella *)
				MB_BitStato[40]:=ModBus.MB_MASTER.ReceiveBuffer.Data[8].0; (*Vedi Tabella *)
				MB_BitStato[41]:=ModBus.MB_MASTER.ReceiveBuffer.Data[8].1; (*Vedi Tabella *)
				MB_BitStato[42]:=ModBus.MB_MASTER.ReceiveBuffer.Data[8].2; (*Vedi Tabella *)
				MB_BitStato[43]:=ModBus.MB_MASTER.ReceiveBuffer.Data[8].3; (*Vedi Tabella *)
				MB_BitStato[44]:=ModBus.MB_MASTER.ReceiveBuffer.Data[8].4; (*Vedi Tabella *)
				MB_BitStato[45]:=ModBus.MB_MASTER.ReceiveBuffer.Data[8].5; (*Vedi Tabella *)
				MB_BitStato[46]:=ModBus.MB_MASTER.ReceiveBuffer.Data[8].6; (*Vedi Tabella *)
				MB_BitStato[47]:=ModBus.MB_MASTER.ReceiveBuffer.Data[8].7; (*Vedi Tabella *)
				MB_BitStato[48]:=ModBus.MB_MASTER.ReceiveBuffer.Data[9].0; (*Vedi Tabella *)
				MB_BitStato[49]:=ModBus.MB_MASTER.ReceiveBuffer.Data[9].1; (*Vedi Tabella *)
				MB_BitStato[50]:=ModBus.MB_MASTER.ReceiveBuffer.Data[9].2; (*Vedi Tabella *)
				MB_BitStato[51]:=ModBus.MB_MASTER.ReceiveBuffer.Data[9].3; (*Vedi Tabella *)
				MB_BitStato[52]:=ModBus.MB_MASTER.ReceiveBuffer.Data[9].4; (*Vedi Tabella *)
				MB_BitStato[53]:=ModBus.MB_MASTER.ReceiveBuffer.Data[9].5; (*Vedi Tabella *)
				MB_BitStato[54]:=ModBus.MB_MASTER.ReceiveBuffer.Data[9].6; (*Vedi Tabella *)
				MB_BitStato[55]:=ModBus.MB_MASTER.ReceiveBuffer.Data[9].7; (*Vedi Tabella *)
				MB_BitStato[56]:=ModBus.MB_MASTER.ReceiveBuffer.Data[10].0; (*Vedi Tabella *)
				MB_BitStato[57]:=ModBus.MB_MASTER.ReceiveBuffer.Data[10].1; (*Vedi Tabella *)
				MB_BitStato[58]:=ModBus.MB_MASTER.ReceiveBuffer.Data[10].2; (*Vedi Tabella *)
				MB_BitStato[59]:=ModBus.MB_MASTER.ReceiveBuffer.Data[10].3; (*Vedi Tabella *)
				MB_BitStato[60]:=ModBus.MB_MASTER.ReceiveBuffer.Data[10].4; (*Vedi Tabella *)
				MB_BitStato[61]:=ModBus.MB_MASTER.ReceiveBuffer.Data[10].5; (*Vedi Tabella *)
				MB_BitStato[62]:=ModBus.MB_MASTER.ReceiveBuffer.Data[10].6; (*Vedi Tabella *)
				MB_BitStato[63]:=ModBus.MB_MASTER.ReceiveBuffer.Data[10].7; (*Vedi Tabella *)
*)
				state:=170;

			END_IF
		END_IF





	170: (* Rispota Altri paramenti COIL *)
		IF NOT ModBus.MB_Start  THEN

			IF ModBus.MB_MASTER.MB_Error<>0 THEN
				state := 300;
			ELSE
				Modbus.MB_Query.SlaveAddress := Address;
				Modbus.MB_Query.FunctionCode := 1;
				ModBus.MB_Query.Read_StartAddress := 0;	(* richiedo lettura altri Parametri *)
				ModBus.MB_Query.Read_Quantity := 64;
				ModBus.MB_Start := TRUE;

				state:=171;
			END_IF
		END_IF
	171: (* Rispota Altri paramenti *)

		IF NOT ModBus.MB_Start  THEN

			IF ModBus.MB_MASTER.MB_Error<>0 THEN
				state := 300;
			ELSE

				MB_BitStatoCoil[0]:=ModBus.MB_MASTER.ReceiveBuffer.Data[3].0; (*Vedi Tabella *)
				MB_BitStatoCoil[1]:=ModBus.MB_MASTER.ReceiveBuffer.Data[3].1; (*Vedi Tabella *)
				MB_BitStatoCoil[2]:=ModBus.MB_MASTER.ReceiveBuffer.Data[3].2; (*Vedi Tabella *)
				MB_BitStatoCoil[3]:=ModBus.MB_MASTER.ReceiveBuffer.Data[3].3; (*Vedi Tabella *)
				MB_BitStatoCoil[4]:=ModBus.MB_MASTER.ReceiveBuffer.Data[3].4; (*Vedi Tabella *)
				MB_BitStatoCoil[5]:=ModBus.MB_MASTER.ReceiveBuffer.Data[3].5; (*Vedi Tabella *)
				MB_BitStatoCoil[6]:=ModBus.MB_MASTER.ReceiveBuffer.Data[3].6; (*Vedi Tabella *)
				MB_BitStatoCoil[7]:=ModBus.MB_MASTER.ReceiveBuffer.Data[3].7; (*Vedi Tabella *)
				MB_BitStatoCoil[8]:=ModBus.MB_MASTER.ReceiveBuffer.Data[4].0; (*Vedi Tabella *)
				MB_BitStatoCoil[9]:=ModBus.MB_MASTER.ReceiveBuffer.Data[4].1; (*Vedi Tabella *)
				MB_BitStatoCoil[10]:=ModBus.MB_MASTER.ReceiveBuffer.Data[4].2; (*Vedi Tabella *)
				MB_BitStatoCoil[11]:=ModBus.MB_MASTER.ReceiveBuffer.Data[4].3; (*Vedi Tabella *)
				MB_BitStatoCoil[12]:=ModBus.MB_MASTER.ReceiveBuffer.Data[4].4; (*Vedi Tabella *)
				MB_BitStatoCoil[13]:=ModBus.MB_MASTER.ReceiveBuffer.Data[4].5; (*Vedi Tabella *)
				MB_BitStatoCoil[14]:=ModBus.MB_MASTER.ReceiveBuffer.Data[4].6; (*Vedi Tabella *)
				MB_BitStatoCoil[15]:=ModBus.MB_MASTER.ReceiveBuffer.Data[4].7; (*Vedi Tabella *)
				MB_BitStatoCoil[16]:=ModBus.MB_MASTER.ReceiveBuffer.Data[5].0; (*Vedi Tabella *)
				MB_BitStatoCoil[17]:=ModBus.MB_MASTER.ReceiveBuffer.Data[5].1; (*Vedi Tabella *)
				MB_BitStatoCoil[18]:=ModBus.MB_MASTER.ReceiveBuffer.Data[5].2; (*Vedi Tabella *)
				MB_BitStatoCoil[19]:=ModBus.MB_MASTER.ReceiveBuffer.Data[5].3; (*Vedi Tabella *)
				MB_BitStatoCoil[20]:=ModBus.MB_MASTER.ReceiveBuffer.Data[5].4; (*Vedi Tabella *)
				MB_BitStatoCoil[21]:=ModBus.MB_MASTER.ReceiveBuffer.Data[5].5; (*Vedi Tabella *)
				MB_BitStatoCoil[22]:=ModBus.MB_MASTER.ReceiveBuffer.Data[5].6; (*Vedi Tabella *)
				MB_BitStatoCoil[23]:=ModBus.MB_MASTER.ReceiveBuffer.Data[5].7; (*Vedi Tabella *)
				MB_BitStatoCoil[24]:=ModBus.MB_MASTER.ReceiveBuffer.Data[6].0; (*Vedi Tabella *)
				MB_BitStatoCoil[25]:=ModBus.MB_MASTER.ReceiveBuffer.Data[6].1; (*Vedi Tabella *)
				MB_BitStatoCoil[26]:=ModBus.MB_MASTER.ReceiveBuffer.Data[6].2; (*Vedi Tabella *)
				MB_BitStatoCoil[27]:=ModBus.MB_MASTER.ReceiveBuffer.Data[6].3; (*Vedi Tabella *)
				MB_BitStatoCoil[28]:=ModBus.MB_MASTER.ReceiveBuffer.Data[6].4; (*Vedi Tabella *)
				MB_BitStatoCoil[29]:=ModBus.MB_MASTER.ReceiveBuffer.Data[6].5; (*Vedi Tabella *)
				MB_BitStatoCoil[30]:=ModBus.MB_MASTER.ReceiveBuffer.Data[6].6; (*Vedi Tabella *)
				MB_BitStatoCoil[31]:=ModBus.MB_MASTER.ReceiveBuffer.Data[6].7; (*Vedi Tabella *)
				MB_BitStatoCoil[32]:=ModBus.MB_MASTER.ReceiveBuffer.Data[7].0; (*Vedi Tabella *)
				MB_BitStatoCoil[33]:=ModBus.MB_MASTER.ReceiveBuffer.Data[7].1; (*Vedi Tabella *)
				MB_BitStatoCoil[34]:=ModBus.MB_MASTER.ReceiveBuffer.Data[7].2; (*Vedi Tabella *)
				MB_BitStatoCoil[35]:=ModBus.MB_MASTER.ReceiveBuffer.Data[7].3; (*Vedi Tabella *)
				MB_BitStatoCoil[36]:=ModBus.MB_MASTER.ReceiveBuffer.Data[7].4; (*Vedi Tabella *)
				MB_BitStatoCoil[37]:=ModBus.MB_MASTER.ReceiveBuffer.Data[7].5; (*Vedi Tabella *)
				MB_BitStatoCoil[38]:=ModBus.MB_MASTER.ReceiveBuffer.Data[7].6; (*Vedi Tabella *)
				MB_BitStatoCoil[39]:=ModBus.MB_MASTER.ReceiveBuffer.Data[7].7; (*Vedi Tabella *)
				MB_BitStatoCoil[40]:=ModBus.MB_MASTER.ReceiveBuffer.Data[8].0; (*Vedi Tabella *)
				MB_BitStatoCoil[41]:=ModBus.MB_MASTER.ReceiveBuffer.Data[8].1; (*Vedi Tabella *)
				MB_BitStatoCoil[42]:=ModBus.MB_MASTER.ReceiveBuffer.Data[8].2; (*Vedi Tabella *)
				MB_BitStatoCoil[43]:=ModBus.MB_MASTER.ReceiveBuffer.Data[8].3; (*Vedi Tabella *)
				MB_BitStatoCoil[44]:=ModBus.MB_MASTER.ReceiveBuffer.Data[8].4; (*Vedi Tabella *)
				MB_BitStatoCoil[45]:=ModBus.MB_MASTER.ReceiveBuffer.Data[8].5; (*Vedi Tabella *)
				MB_BitStatoCoil[46]:=ModBus.MB_MASTER.ReceiveBuffer.Data[8].6; (*Vedi Tabella *)
				MB_BitStatoCoil[47]:=ModBus.MB_MASTER.ReceiveBuffer.Data[8].7; (*Vedi Tabella *)
				MB_BitStatoCoil[48]:=ModBus.MB_MASTER.ReceiveBuffer.Data[9].0; (*Vedi Tabella *)
				MB_BitStatoCoil[49]:=ModBus.MB_MASTER.ReceiveBuffer.Data[9].1; (*Vedi Tabella *)
				MB_BitStatoCoil[50]:=ModBus.MB_MASTER.ReceiveBuffer.Data[9].2; (*Vedi Tabella *)
				MB_BitStatoCoil[51]:=ModBus.MB_MASTER.ReceiveBuffer.Data[9].3; (*Vedi Tabella *)
				MB_BitStatoCoil[52]:=ModBus.MB_MASTER.ReceiveBuffer.Data[9].4; (*Vedi Tabella *)
				MB_BitStatoCoil[53]:=ModBus.MB_MASTER.ReceiveBuffer.Data[9].5; (*Vedi Tabella *)
				MB_BitStatoCoil[54]:=ModBus.MB_MASTER.ReceiveBuffer.Data[9].6; (*Vedi Tabella *)
				MB_BitStatoCoil[55]:=ModBus.MB_MASTER.ReceiveBuffer.Data[9].7; (*Vedi Tabella *)
				MB_BitStatoCoil[56]:=ModBus.MB_MASTER.ReceiveBuffer.Data[10].0; (*Vedi Tabella *)
				MB_BitStatoCoil[57]:=ModBus.MB_MASTER.ReceiveBuffer.Data[10].1; (*Vedi Tabella *)
				MB_BitStatoCoil[58]:=ModBus.MB_MASTER.ReceiveBuffer.Data[10].2; (*Vedi Tabella *)
				MB_BitStatoCoil[59]:=ModBus.MB_MASTER.ReceiveBuffer.Data[10].3; (*Vedi Tabella *)
				MB_BitStatoCoil[60]:=ModBus.MB_MASTER.ReceiveBuffer.Data[10].4; (*Vedi Tabella *)
				MB_BitStatoCoil[61]:=ModBus.MB_MASTER.ReceiveBuffer.Data[10].5; (*Vedi Tabella *)
				MB_BitStatoCoil[62]:=ModBus.MB_MASTER.ReceiveBuffer.Data[10].6; (*Vedi Tabella *)
				MB_BitStatoCoil[63]:=ModBus.MB_MASTER.ReceiveBuffer.Data[10].7; (*Vedi Tabella *)
				MB_BitStatoCoil[64]:=ModBus.MB_MASTER.ReceiveBuffer.Data[11].0; (*Vedi Tabella *)
				MB_BitStatoCoil[65]:=ModBus.MB_MASTER.ReceiveBuffer.Data[11].1; (*Vedi Tabella *)
				MB_BitStatoCoil[66]:=ModBus.MB_MASTER.ReceiveBuffer.Data[1].2; (*Vedi Tabella *)
				MB_BitStatoCoil[67]:=ModBus.MB_MASTER.ReceiveBuffer.Data[11].3; (*Vedi Tabella *)
				MB_BitStatoCoil[68]:=ModBus.MB_MASTER.ReceiveBuffer.Data[11].4; (*Vedi Tabella *)
				MB_BitStatoCoil[69]:=ModBus.MB_MASTER.ReceiveBuffer.Data[11].5; (*Vedi Tabella *)
				MB_BitStatoCoil[70]:=ModBus.MB_MASTER.ReceiveBuffer.Data[11].6; (*Vedi Tabella *)
				MB_BitStatoCoil[71]:=ModBus.MB_MASTER.ReceiveBuffer.Data[11].7; (*Vedi Tabella *)
				state:=190 ;   (**********************************************************************************************************************+******)

			END_IF
		END_IF

		190:    (* Scrittura BOOL - COIL o WORD *)
		IF NOT ModBus.MB_Start THEN
			IF ModBus.MB_MASTER.MB_Error<>0 THEN (*OR ModBus.MB_MASTER.MB_Error<>0 THEN*)
				state := 300;
			ELSE
				IF ScriviDato THEN
					IF ScriviCoil THEN
						Modbus.MB_Query.FunctionCode := 5;
					ELSE
						Modbus.MB_Query.FunctionCode := 6;
					END_IF
					Modbus.MB_Query.SlaveAddress := Address;
					ModBus.MB_Query.Write_StartAddress := IndirizzoDaScrivere;
					ModBus.MB_Query.Write_Quantity :=1;
					ModBus.MB_Query.Write_Data[0] := DatoDaScrivere;
					ModBus.MB_Start := TRUE;
						IF Test_ScriviCoil THEN
							IF 	MB_BitStatoCoil[IndirizzoDaScrivere]=WORD_TO_BOOL(DatoDaScrivere) THEN
								ScriviDato:=FALSE;
							END_IF
						ELSE
							IF 	MB_RegistriHoldingLetti[IndirizzoDaScrivere]=DatoDaScrivere THEN
								ScriviDato:=FALSE;
							END_IF
						END_IF
					state := 200;
				ELSE
					state := 200;
				END_IF
			END_IF
		END_IF



		200:    (* Scrittura BOOL Abilita UTA 01 *)
		IF NOT ModBus.MB_Start THEN
			IF ModBus.MB_MASTER.MB_Error<>0 THEN (*OR ModBus.MB_MASTER.MB_Error<>0 THEN*)
				state := 300;
			ELSE
				IF ControlMode_UTA01   THEN
					Modbus.MB_Query.FunctionCode := 5;
					Modbus.MB_Query.SlaveAddress := Address;
					ModBus.MB_Query.Write_StartAddress := 19;
					ModBus.MB_Query.Write_Quantity :=1;
					ModBus.MB_Query.Write_Data[0] := BOOL_TO_WORD(ScriviRUN_UTA01);
					ModBus.MB_Start := TRUE;
					state := 202;
				ELSE
					state := 202;
				END_IF
			END_IF
		END_IF

		202:    (* Scrittura Set Point  UTA 01 *)
		IF NOT ModBus.MB_Start THEN
			IF ModBus.MB_MASTER.MB_Error<>0 THEN (*OR ModBus.MB_MASTER.MB_Error<>0 THEN*)
				state := 300;
			ELSE
				IF ControlMode_UTA01   THEN
					Modbus.MB_Query.FunctionCode :=6;
					Modbus.MB_Query.SlaveAddress := Address;
					ModBus.MB_Query.Write_StartAddress := 69;
					ModBus.MB_Query.Write_Quantity :=1;
					ModBus.MB_Query.Write_Data[0] :=ScriviSP_UTA01;
					ModBus.MB_Start := TRUE;
					state := 205;
				ELSE
					state := 205;
				END_IF
			END_IF
		END_IF

		205:    (* Scrittura BOOL Abilita UTA 02 *)
		IF NOT ModBus.MB_Start THEN
			IF ModBus.MB_MASTER.MB_Error<>0 THEN (*OR ModBus.MB_MASTER.MB_Error<>0 THEN*)
				state := 300;
			ELSE
				IF ControlMode_UTA02   THEN
					Modbus.MB_Query.FunctionCode := 5;
					Modbus.MB_Query.SlaveAddress := Address;
					ModBus.MB_Query.Write_StartAddress := 20;
					ModBus.MB_Query.Write_Quantity :=1;
					ModBus.MB_Query.Write_Data[0] := BOOL_TO_WORD(ScriviRUN_UTA02);
					ModBus.MB_Start := TRUE;
					state := 206;
				ELSE
					state := 206;
				END_IF
			END_IF
		END_IF

		206:    (* Scrittura Set Point  UTA 02 *)
		IF NOT ModBus.MB_Start THEN
			IF ModBus.MB_MASTER.MB_Error<>0 THEN (*OR ModBus.MB_MASTER.MB_Error<>0 THEN*)
				state := 300;
			ELSE
				IF  ControlMode_UTA02 THEN
					Modbus.MB_Query.FunctionCode :=6;
					Modbus.MB_Query.SlaveAddress := Address;
					ModBus.MB_Query.Write_StartAddress := 79;
					ModBus.MB_Query.Write_Quantity :=1;
					ModBus.MB_Query.Write_Data[0] :=ScriviSP_UTA02;
					ModBus.MB_Start := TRUE;
					state := 210;
				ELSE
					state := 210;
				END_IF
			END_IF
		END_IF

		210:    (* Scrittura BOOL Abilita UTA 03 *)
		IF NOT ModBus.MB_Start THEN
			IF ModBus.MB_MASTER.MB_Error<>0 THEN (*OR ModBus.MB_MASTER.MB_Error<>0 THEN*)
				state := 300;
			ELSE
				IF ControlMode_UTA03   THEN
					Modbus.MB_Query.FunctionCode := 5;
					Modbus.MB_Query.SlaveAddress := Address;
					ModBus.MB_Query.Write_StartAddress := 21;
					ModBus.MB_Query.Write_Quantity :=1;
					ModBus.MB_Query.Write_Data[0] := BOOL_TO_WORD(ScriviRUN_UTA03);
					ModBus.MB_Start := TRUE;
					state := 211;
				ELSE
					state := 211;
				END_IF
			END_IF
		END_IF

		211:    (* Scrittura Set Point  UTA 03 *)
		IF NOT ModBus.MB_Start THEN
			IF ModBus.MB_MASTER.MB_Error<>0 THEN (*OR ModBus.MB_MASTER.MB_Error<>0 THEN*)
				state := 300;
			ELSE
				IF ControlMode_UTA03  THEN
					Modbus.MB_Query.FunctionCode :=6;
					Modbus.MB_Query.SlaveAddress := Address;
					ModBus.MB_Query.Write_StartAddress := 88;
					ModBus.MB_Query.Write_Quantity :=1;
					ModBus.MB_Query.Write_Data[0] :=ScriviSP_UTA03;
					ModBus.MB_Start := TRUE;
					state := 215;
				ELSE
					state := 215;
				END_IF
			END_IF
		END_IF

		215:    (* Scrittura BOOL Abilita UTA 04 *)
		IF NOT ModBus.MB_Start THEN
			IF ModBus.MB_MASTER.MB_Error<>0 THEN (*OR ModBus.MB_MASTER.MB_Error<>0 THEN*)
				state := 300;
			ELSE
				IF ControlMode_UTA04   THEN
					Modbus.MB_Query.FunctionCode := 5;
					Modbus.MB_Query.SlaveAddress := Address;
					ModBus.MB_Query.Write_StartAddress := 22;
					ModBus.MB_Query.Write_Quantity :=1;
					ModBus.MB_Query.Write_Data[0] := BOOL_TO_WORD(ScriviRUN_UTA04);
					ModBus.MB_Start := TRUE;
					state := 216;
				ELSE
					state := 216;
				END_IF
			END_IF
		END_IF

		216:    (* Scrittura Set Point  UTA 04 *)
		IF NOT ModBus.MB_Start THEN
			IF ModBus.MB_MASTER.MB_Error<>0 THEN (*OR ModBus.MB_MASTER.MB_Error<>0 THEN*)
				state := 300;
			ELSE
				IF ControlMode_UTA04  THEN
					Modbus.MB_Query.FunctionCode :=6;
					Modbus.MB_Query.SlaveAddress := Address;
					ModBus.MB_Query.Write_StartAddress := 99;
					ModBus.MB_Query.Write_Quantity :=1;
					ModBus.MB_Query.Write_Data[0] :=ScriviSP_UTA04;
					ModBus.MB_Start := TRUE;
					state := 220;
				ELSE
					state := 220;
				END_IF
			END_IF
		END_IF

		220:    (* Scrittura BOOL Abilita UTA 05 *)
		IF NOT ModBus.MB_Start THEN
			IF ModBus.MB_MASTER.MB_Error<>0 THEN (*OR ModBus.MB_MASTER.MB_Error<>0 THEN*)
				state := 300;
			ELSE
				IF ControlMode_UTA05   THEN
					Modbus.MB_Query.FunctionCode := 5;
					Modbus.MB_Query.SlaveAddress := Address;
					ModBus.MB_Query.Write_StartAddress := 23;
					ModBus.MB_Query.Write_Quantity :=1;
					ModBus.MB_Query.Write_Data[0] := BOOL_TO_WORD(ScriviRUN_UTA05);
					ModBus.MB_Start := TRUE;
					state := 221;
				ELSE
					state := 221;
				END_IF
			END_IF
		END_IF

		221:    (* Scrittura Set Point  UTA 05 *)
		IF NOT ModBus.MB_Start THEN
			IF ModBus.MB_MASTER.MB_Error<>0 THEN (*OR ModBus.MB_MASTER.MB_Error<>0 THEN*)
				state := 300;
			ELSE
				IF ControlMode_UTA05  THEN
					Modbus.MB_Query.FunctionCode :=6;
					Modbus.MB_Query.SlaveAddress := Address;
					ModBus.MB_Query.Write_StartAddress :=108;
					ModBus.MB_Query.Write_Quantity :=1;
					ModBus.MB_Query.Write_Data[0] :=ScriviSP_UTA05;
					ModBus.MB_Start := TRUE;
					state := 225;
				ELSE
					state := 225;
				END_IF
			END_IF
		END_IF

		225:    (* Scrittura BOOL Abilita UTA 06 *)
		IF NOT ModBus.MB_Start THEN
			IF ModBus.MB_MASTER.MB_Error<>0 THEN (*OR ModBus.MB_MASTER.MB_Error<>0 THEN*)
				state := 300;
			ELSE
				IF ControlMode_UTA06   THEN
					Modbus.MB_Query.FunctionCode := 5;
					Modbus.MB_Query.SlaveAddress := Address;
					ModBus.MB_Query.Write_StartAddress := 1;
					ModBus.MB_Query.Write_Quantity :=1;
					ModBus.MB_Query.Write_Data[0] := BOOL_TO_WORD(ScriviRUN_UTA06);
					ModBus.MB_Start := TRUE;
					state := 226;
				ELSE
					state := 226;
				END_IF
			END_IF
		END_IF

		226:    (* Scrittura Set Point  UTA 06 *)
		IF NOT ModBus.MB_Start THEN
			IF ModBus.MB_MASTER.MB_Error<>0 THEN (*OR ModBus.MB_MASTER.MB_Error<>0 THEN*)
				state := 300;
			ELSE
				IF ControlMode_UTA06  THEN
					Modbus.MB_Query.FunctionCode :=6;
					Modbus.MB_Query.SlaveAddress := Address;
					ModBus.MB_Query.Write_StartAddress := 1;
					ModBus.MB_Query.Write_Quantity :=1;
					ModBus.MB_Query.Write_Data[0] :=ScriviSP_UTA06;
					ModBus.MB_Start := TRUE;
					state := 230;
				ELSE
					state := 230;
				END_IF
			END_IF
		END_IF

		230:    (* Scrittura BOOL Abilita UTA 07 *)
		IF NOT ModBus.MB_Start THEN
			IF ModBus.MB_MASTER.MB_Error<>0 THEN (*OR ModBus.MB_MASTER.MB_Error<>0 THEN*)
				state := 300;
			ELSE
				IF ControlMode_UTA07  THEN
					Modbus.MB_Query.FunctionCode := 5;
					Modbus.MB_Query.SlaveAddress := Address;
					ModBus.MB_Query.Write_StartAddress := 2;
					ModBus.MB_Query.Write_Quantity :=1;
					ModBus.MB_Query.Write_Data[0] := BOOL_TO_WORD(ScriviRUN_UTA07);
					ModBus.MB_Start := TRUE;
					state := 231;
				ELSE
					state := 231;
				END_IF
			END_IF
		END_IF

		231:    (* Scrittura Set Point  UTA 07 *)
		IF NOT ModBus.MB_Start THEN
			IF ModBus.MB_MASTER.MB_Error<>0 THEN (*OR ModBus.MB_MASTER.MB_Error<>0 THEN*)
				state := 300;
			ELSE
				IF ControlMode_UTA07  THEN
					Modbus.MB_Query.FunctionCode :=6;
					Modbus.MB_Query.SlaveAddress := Address;
					ModBus.MB_Query.Write_StartAddress :=11;
					ModBus.MB_Query.Write_Quantity :=1;
					ModBus.MB_Query.Write_Data[0] :=ScriviSP_UTA07;
					ModBus.MB_Start := TRUE;
					state := 235;
				ELSE
					state := 235;
				END_IF
			END_IF
		END_IF

		235:    (* Scrittura BOOL Abilita UTA 08 *)
		IF NOT ModBus.MB_Start THEN
			IF ModBus.MB_MASTER.MB_Error<>0 THEN (*OR ModBus.MB_MASTER.MB_Error<>0 THEN*)
				state := 300;
			ELSE
				IF ControlMode_UTA08  THEN
					Modbus.MB_Query.FunctionCode := 5;
					Modbus.MB_Query.SlaveAddress := Address;
					ModBus.MB_Query.Write_StartAddress := 10;
					ModBus.MB_Query.Write_Quantity :=1;
					ModBus.MB_Query.Write_Data[0] := BOOL_TO_WORD(ScriviRUN_UTA08);
					ModBus.MB_Start := TRUE;
					state := 236;
				ELSE
					state := 236;
				END_IF
			END_IF
		END_IF

		236:    (* Scrittura Set Point  UTA 08 *)
		IF NOT ModBus.MB_Start THEN
			IF ModBus.MB_MASTER.MB_Error<>0 THEN (*OR ModBus.MB_MASTER.MB_Error<>0 THEN*)
				state := 300;
			ELSE
				IF ControlMode_UTA08  THEN
					Modbus.MB_Query.FunctionCode :=6;
					Modbus.MB_Query.SlaveAddress := Address;
					ModBus.MB_Query.Write_StartAddress := 25;
					ModBus.MB_Query.Write_Quantity :=1;
					ModBus.MB_Query.Write_Data[0] :=ScriviSP_UTA08;
					ModBus.MB_Start := TRUE;
					state := 240;
				ELSE
					state := 240;
				END_IF
			END_IF
		END_IF

		240:    (* Scrittura BOOL Abilita UTA 09 *)
		IF NOT ModBus.MB_Start THEN
			IF ModBus.MB_MASTER.MB_Error<>0 THEN (*OR ModBus.MB_MASTER.MB_Error<>0 THEN*)
				state := 300;
			ELSE
				IF ControlMode_UTA09  THEN
					Modbus.MB_Query.FunctionCode := 5;
					Modbus.MB_Query.SlaveAddress := Address;
					ModBus.MB_Query.Write_StartAddress :=11;
					ModBus.MB_Query.Write_Quantity :=1;
					ModBus.MB_Query.Write_Data[0] := BOOL_TO_WORD(ScriviRUN_UTA09);
					ModBus.MB_Start := TRUE;
					state := 241;
				ELSE
					state := 241;
				END_IF
			END_IF
		END_IF

		241:    (* Scrittura Set Point  UTA 09 *)
		IF NOT ModBus.MB_Start THEN
			IF ModBus.MB_MASTER.MB_Error<>0 THEN (*OR ModBus.MB_MASTER.MB_Error<>0 THEN*)
				state := 300;
			ELSE
				IF ControlMode_UTA09  THEN
					Modbus.MB_Query.FunctionCode :=6;
					Modbus.MB_Query.SlaveAddress := Address;
					ModBus.MB_Query.Write_StartAddress :=35;
					ModBus.MB_Query.Write_Quantity :=1;
					ModBus.MB_Query.Write_Data[0] :=ScriviSP_UTA09;
					ModBus.MB_Start := TRUE;
					state := 245;
				ELSE
					state := 245;
				END_IF
			END_IF
		END_IF

		245:    (* Scrittura BOOL Abilita UTA10 *)
		IF NOT ModBus.MB_Start THEN
			IF ModBus.MB_MASTER.MB_Error<>0 THEN (*OR ModBus.MB_MASTER.MB_Error<>0 THEN*)
				state := 300;
			ELSE
				IF ControlMode_UTA10  THEN
					Modbus.MB_Query.FunctionCode := 5;
					Modbus.MB_Query.SlaveAddress := Address;
					ModBus.MB_Query.Write_StartAddress := 65;
					ModBus.MB_Query.Write_Quantity :=1;
					ModBus.MB_Query.Write_Data[0] := BOOL_TO_WORD(ScriviRUN_UTA10);
					ModBus.MB_Start := TRUE;
					state := 246;
				ELSE
					state := 246;
				END_IF
			END_IF
		END_IF

		246:    (* Scrittura Set Point  UTA 10 *)
		IF NOT ModBus.MB_Start THEN
			IF ModBus.MB_MASTER.MB_Error<>0 THEN (*OR ModBus.MB_MASTER.MB_Error<>0 THEN*)
				state := 300;
			ELSE
				IF ControlMode_UTA10  THEN
					Modbus.MB_Query.FunctionCode :=6;
					Modbus.MB_Query.SlaveAddress := Address;
					ModBus.MB_Query.Write_StartAddress := 160;
					ModBus.MB_Query.Write_Quantity :=1;
					ModBus.MB_Query.Write_Data[0] :=ScriviSP_UTA10;
					ModBus.MB_Start := TRUE;
					state := 250;
				ELSE
					state := 250;
				END_IF
			END_IF
		END_IF

		250:    (* Scrittura BOOL Abilita UTA 11  NON PRESENTE  *)
		IF NOT ModBus.MB_Start THEN
			IF ModBus.MB_MASTER.MB_Error<>0 THEN (*OR ModBus.MB_MASTER.MB_Error<>0 THEN*)
				state := 300;
			ELSE
				state := 255;
			END_IF
		END_IF



		255:    (* Scrittura BOOL Abilita UTA12 *)
		IF NOT ModBus.MB_Start THEN
			IF ModBus.MB_MASTER.MB_Error<>0 THEN (*OR ModBus.MB_MASTER.MB_Error<>0 THEN*)
				state := 300;
			ELSE
				IF ControlMode_UTA12  THEN
					Modbus.MB_Query.FunctionCode := 5;
					Modbus.MB_Query.SlaveAddress := Address;
					ModBus.MB_Query.Write_StartAddress := 14;
					ModBus.MB_Query.Write_Quantity :=1;
					ModBus.MB_Query.Write_Data[0] := BOOL_TO_WORD(ScriviRUN_UTA12);
					ModBus.MB_Start := TRUE;
					state := 256;
				ELSE
					state := 256;
				END_IF
			END_IF
		END_IF

		256:    (* Scrittura Set Point  UTA 12 *)
		IF NOT ModBus.MB_Start THEN
			IF ModBus.MB_MASTER.MB_Error<>0 THEN (*OR ModBus.MB_MASTER.MB_Error<>0 THEN*)
				state := 300;
			ELSE
				IF ControlMode_UTA12  THEN
					Modbus.MB_Query.FunctionCode :=6;
					Modbus.MB_Query.SlaveAddress := Address;
					ModBus.MB_Query.Write_StartAddress := 53;
					ModBus.MB_Query.Write_Quantity :=1;
					ModBus.MB_Query.Write_Data[0] :=ScriviSP_UTA12;
					ModBus.MB_Start := TRUE;
					state := 260;
				ELSE
					state := 260;
				END_IF
			END_IF
		END_IF



		260:    (* Scrittura BOOL Abilita UTA 13 *)
		IF NOT ModBus.MB_Start THEN
			IF ModBus.MB_MASTER.MB_Error<>0 THEN (*OR ModBus.MB_MASTER.MB_Error<>0 THEN*)
				state := 300;
			ELSE
				IF ControlMode_UTA13  THEN
					Modbus.MB_Query.FunctionCode := 5;
					Modbus.MB_Query.SlaveAddress := Address;
					ModBus.MB_Query.Write_StartAddress :=18;
					ModBus.MB_Query.Write_Quantity :=1;
					ModBus.MB_Query.Write_Data[0] := BOOL_TO_WORD(ScriviRUN_UTA13);
					ModBus.MB_Start := TRUE;
					state := 261;
				ELSE
					state := 261;
				END_IF
			END_IF
		END_IF

		261:    (* Scrittura Set Point  UTA 13 *)
		IF NOT ModBus.MB_Start THEN
			IF ModBus.MB_MASTER.MB_Error<>0 THEN (*OR ModBus.MB_MASTER.MB_Error<>0 THEN*)
				state := 300;
			ELSE
				IF ControlMode_UTA13  THEN
					Modbus.MB_Query.FunctionCode :=6;
					Modbus.MB_Query.SlaveAddress := Address;
					ModBus.MB_Query.Write_StartAddress :=64;
					ModBus.MB_Query.Write_Quantity :=1;
					ModBus.MB_Query.Write_Data[0] :=ScriviSP_UTA13;
					ModBus.MB_Start := TRUE;
					state := 295;
				ELSE
					state := 295;
				END_IF
			END_IF
		END_IF

		295:
		IF NOT ModBus.MB_Start THEN
			IF ModBus.MB_MASTER.MB_Error<>0 THEN (*OR ModBus.MB_MASTER.MB_Error<>0 THEN*)
				state := 300;
			ELSE
				IF fModbusAlr THEN fModbusAlr := FALSE; END_IF
				NodoDaInterrogareANZ:=Address+1;
				InibiscoModbusANZ:=FALSE;
				retryErr := 0;
				retry := 0;
				state := 0;
					IF fModbusAlr=FALSE AND ErroreComuModBus=TRUE THEN
						LogEv(EL_Log,EO_CHI,ID,62,'ComunicazioneModBus_OK');
						ErroreComuModBus := FALSE;
				(*	WarningCtr := SEL(WarningCtr=0, WarningCtr-1, 0); *)
					END_IF


			END_IF
		END_IF



	(**** CHECK MODBUS ERROR ****)
	300: 	(* Release MODBUS *)
			InibiscoModbusMB1:=FALSE;
			(* Retries *)
			retry:=retry+1;
			IF retry>3 THEN
				retry:=0;

				(* Verify if slave is dead *)
				IF retryErr < retryErrMaX THEN
					retryErr := retryErr + 1;
				ELSE
					fModbusAlr := TRUE;
					(* Verify ModBus error	*)

					IF fModbusAlr AND ErroreComuModBus=FALSE THEN
						LogEv(EL_Alarm,EO_CHI,ID,61,CONCAT('ErroreModbus_',INT_TO_STRING(ModBus.MB_MASTER.MB_Error)));
						ErroreComuModBus := TRUE;
					END_IF
				END_IF

				END_IF
			Refresh_Now := FALSE;
			InibiscoModbusMB1:=FALSE;
			NodoDaInterrogareMB1:=Address;
			state:=0;
END_CASE




(* Controllo Time Out Ciclo ModBus *)

TimeOutModBus(In:=state<>0,PT:=t#30s);
IF TimeOutModBus.Q THEN
	State:=0;

	IF MODBUS.MB_Lock=TRUE THEN MODBUS.MB_Lock:=FALSE;END_IF
	IF InibiscoModbusMB1=TRUE THEN InibiscoModbusMB1:=FALSE;END_IF
END_IF
END_ACTION

(* POU Plant_Objects/obj_UTA_02, ST *)
FUNCTION_BLOCK obj_UTA_02
VAR_INPUT
	ID				: BYTE;

	UTA_ST : BOOL;
	UTA_CentrAL : BOOL;
	UTA_CONTROL_MODE:BOOL:=FALSE;

	(* Physical inputs (Force) *)
	UTA_RUN_REQ		: BOOL; (* External run request (no heat or cold requested) *)
	UTA_STOP_REQ	: BOOL; (* External stop request (has priority over RUN signals!) *)



	cmd_DI_RUN: BOOL;		(* variabili di appoggio per avviare l'UTA in locale, poi verrà trasferito ad un OUT per essere passato al Bloco trend *)
	cmd_DI_SetPoint: INT;		(* variabili di appoggio per avviare l'UTA in locale, poi verrà trasferito ad un OUT per essere passato al Bloco trend *)

	T_AMB: INT;
	UR_AMB: INT;
	T_MISC: INT;
	UR_MISC: INT;
	T_MAND: INT;
	T_EST: INT;
	UR_EST: INT;
	ENTALPIA_EST: INT;
	ENTALPIA_AMB: INT;
	UMID_ASS_EST: INT;
	UMID_ASS_AMB: INT;
	UMID_ASS_MISC: INT;
	UMID_ASS_CONDEN: INT;
	SET_COMP_T_AMB: INT;
	RITAR_SET_T_AMB: INT;
	SET_T_MAND: INT;
	SET_ANTIGELO: INT;
	SET_UR_AMB: INT;
	ISTERESI_UR_AMB: INT;
	SET_F_ANTIG_AMB: INT;
	SOGLIA_T_EST_VR: INT;
	MIN_AP_SERR_E_R: INT;
	MIN_AP_SERR_ESP: INT;
	RID_SET_T_RISC: INT;
	VENT_MAND: BOOL;
	VENT_RIPR: BOOL;
	P_UMIDIF: BOOL;
	VALV_B_FREDDA: BOOL;
	VALV_B_CALDA: BOOL;
	SERRANDE_ESP: BOOL;
	SERRAND_EST_RIC: BOOL;
	ABILITA: BOOL;
	STATO_VENT_M: BOOL;
	STATO_VENT_R: BOOL;
	FILTRO: BOOL;
	FLUSSO_VM: BOOL;
	FLUSSO_VR: BOOL;
	FILTRI_INTASATI: BOOL;
	ALL_VERIFICA_VM: BOOL;
	ALL_VERIFICA_VR: BOOL;
	ALL_V011_MANC_SPEGN: BOOL;
	ALL_V011_MANC_FUNZ: BOOL;
	ALL_V012_MANC_SPEGN: BOOL;
	ALL_V012_MANC_FUNZ: BOOL;


END_VAR
VAR_OUTPUT

	cmd_DO_OUT: BOOL;
	cmd_DO_SetPoint:INT;

END_VAR
VAR

	Status_Log		: WORD;
	Status_Vis		: DWORD;


	AllarmeScattoTermico: BOOL;
	AlarmHw		:	FLT_TAP := (INITEV:=FALSE);

(* per creazione stringa da loggare ***)
	temp :STRING(255);
	tempRaw		: ARRAY [0..MAX_SEND_TCP_CLIENT] OF BYTE;
	tempRawLen :DINT;
	longString:STRING(800);



	moreno: STRING;
END_VAR
	IF UTA_STOP_REQ THEN cmd_DO_OUT := FALSE;
		ELSIF UTA_RUN_REQ THEN cmd_DO_OUT := TRUE;
		ELSE cmd_DO_OUT := cmd_DI_RUN  ;
	END_IF

cmd_DO_SetPoint:=cmd_DI_SetPoint;


(* Hardware alarm (physical input *)
AlarmHw(IN:=UTA_CentrAL);     (* TRUE= Flusso , FALSE = No Flusso *)

IF AlarmHw.EVH THEN
	LogEv(EL_Alarm,EO_UTACOIN,ID,3,'UTA_Riarmato');
END_IF

IF AlarmHw.EVL THEN
	LogEv(EL_Log,EO_UTACOIN,ID,4,'AllarmeUTA');
END_IF

AllarmeScattoTermico := NOT UTA_CentrAL;


(* segnalazione Allarme *)
IF AllarmeScattoTermico  THEN
	Status_Log := 2;
	Status_Vis := COLOR_RED;

ELSIF

	ALL_VERIFICA_VM OR
	ALL_VERIFICA_VR OR
	ALL_V011_MANC_SPEGN OR
	ALL_V011_MANC_FUNZ OR
	ALL_V012_MANC_SPEGN OR
	ALL_V012_MANC_FUNZ THEN

	Status_Log := 1;
	Status_Vis := COLOR_YELLOW;


ELSE
	Status_Log := 0;
	Status_Vis := COLOR_GREEN;
END_IF
END_FUNCTION_BLOCK
ACTION AddLogData:
Logger.s1:=INSERT('&UTACOIN=',BYTE_TO_STRING(ID),8);
IF ID<10 THEN Logger.s1:=INSERT(Logger.s1,'0',8); END_IF



(* inizializzo stringa da loggare **)
FOR tempRawLen:=0 TO MAX_SEND_TCP_CLIENT DO
                tempRaw[tempRawLen]:=0;
END_FOR

tempRawLen:=0;


temp:=Logger.s1;
moreno:=Logger.s1;
ADDSTRING(ADR(tempRaw), ADR(temp), tempRawLen);



	temp:=CONCAT(INT_TO_STRING(T_AMB),';'); 						(*  1 *)
	ADDSTRING(ADR(tempRaw), ADR(temp), tempRawLen);
	temp:=CONCAT(INT_TO_STRING(UR_AMB),';');
	ADDSTRING(ADR(tempRaw), ADR(temp), tempRawLen);
	temp:=CONCAT(INT_TO_STRING(T_MISC),';');
	ADDSTRING(ADR(tempRaw), ADR(temp), tempRawLen);
	temp:=CONCAT(INT_TO_STRING(UR_MISC),';');
	ADDSTRING(ADR(tempRaw), ADR(temp), tempRawLen);
	temp:=CONCAT(INT_TO_STRING(T_MAND),';');
	ADDSTRING(ADR(tempRaw), ADR(temp), tempRawLen);
	temp:=CONCAT(INT_TO_STRING(T_EST),';');
	ADDSTRING(ADR(tempRaw), ADR(temp), tempRawLen);
	temp:=CONCAT(INT_TO_STRING(UR_EST),';');
	ADDSTRING(ADR(tempRaw), ADR(temp), tempRawLen);
	temp:=CONCAT(INT_TO_STRING(ENTALPIA_EST),';');
	ADDSTRING(ADR(tempRaw), ADR(temp), tempRawLen);
	temp:=CONCAT(INT_TO_STRING(ENTALPIA_AMB),';');
	ADDSTRING(ADR(tempRaw), ADR(temp), tempRawLen);
	temp:=CONCAT(INT_TO_STRING(UMID_ASS_EST),';');				(*  10 *)
	ADDSTRING(ADR(tempRaw), ADR(temp), tempRawLen);
	temp:=CONCAT(INT_TO_STRING(UMID_ASS_AMB),';');
	ADDSTRING(ADR(tempRaw), ADR(temp), tempRawLen);
	temp:=CONCAT(INT_TO_STRING(UMID_ASS_MISC),';');
	ADDSTRING(ADR(tempRaw), ADR(temp), tempRawLen);
	temp:=CONCAT(INT_TO_STRING(UMID_ASS_CONDEN),';');
	ADDSTRING(ADR(tempRaw), ADR(temp), tempRawLen);
	temp:=CONCAT(INT_TO_STRING(SET_COMP_T_AMB),';');
	ADDSTRING(ADR(tempRaw), ADR(temp), tempRawLen);
	temp:=CONCAT(INT_TO_STRING(RITAR_SET_T_AMB),';');
	ADDSTRING(ADR(tempRaw), ADR(temp), tempRawLen);
	temp:=CONCAT(INT_TO_STRING(SET_T_MAND),';');
	ADDSTRING(ADR(tempRaw), ADR(temp), tempRawLen);
	temp:=CONCAT(INT_TO_STRING(SET_ANTIGELO),';');
	ADDSTRING(ADR(tempRaw), ADR(temp), tempRawLen);
	temp:=CONCAT(INT_TO_STRING(SET_UR_AMB),';');
	ADDSTRING(ADR(tempRaw), ADR(temp), tempRawLen);
	temp:=CONCAT(INT_TO_STRING(ISTERESI_UR_AMB),';');
	ADDSTRING(ADR(tempRaw), ADR(temp), tempRawLen);
	temp:=CONCAT(INT_TO_STRING(SET_F_ANTIG_AMB),';');			(*  20 *)
	ADDSTRING(ADR(tempRaw), ADR(temp), tempRawLen);
	temp:=CONCAT(INT_TO_STRING(SOGLIA_T_EST_VR),';');
	ADDSTRING(ADR(tempRaw), ADR(temp), tempRawLen);
	temp:=CONCAT(INT_TO_STRING(MIN_AP_SERR_E_R),';');
	ADDSTRING(ADR(tempRaw), ADR(temp), tempRawLen);
	temp:=CONCAT(INT_TO_STRING(MIN_AP_SERR_ESP),';');
	ADDSTRING(ADR(tempRaw), ADR(temp), tempRawLen);
	temp:=CONCAT(INT_TO_STRING(RID_SET_T_RISC),';');
	ADDSTRING(ADR(tempRaw), ADR(temp), tempRawLen);


	temp:=CONCAT(SEL(VENT_MAND,'0','1'),';');
	ADDSTRING(ADR(tempRaw), ADR(temp), tempRawLen);
	temp:=CONCAT(SEL(VENT_RIPR,'0','1'),';');
	ADDSTRING(ADR(tempRaw), ADR(temp), tempRawLen);
	temp:=CONCAT(SEL(P_UMIDIF,'0','1'),';');
	ADDSTRING(ADR(tempRaw), ADR(temp), tempRawLen);
	temp:=CONCAT(SEL(VALV_B_FREDDA,'0','1'),';');
	ADDSTRING(ADR(tempRaw), ADR(temp), tempRawLen);
	temp:=CONCAT(SEL(VALV_B_CALDA,'0','1'),';');
	ADDSTRING(ADR(tempRaw), ADR(temp), tempRawLen);
	temp:=CONCAT(SEL(SERRANDE_ESP,'0','1'),';');						(*  30 *)
	ADDSTRING(ADR(tempRaw), ADR(temp), tempRawLen);
	temp:=CONCAT(SEL(SERRAND_EST_RIC,'0','1'),';');
	ADDSTRING(ADR(tempRaw), ADR(temp), tempRawLen);
	temp:=CONCAT(SEL(ABILITA,'0','1'),';');
	ADDSTRING(ADR(tempRaw), ADR(temp), tempRawLen);
	temp:=CONCAT(SEL(STATO_VENT_M,'0','1'),';');
	ADDSTRING(ADR(tempRaw), ADR(temp), tempRawLen);
	temp:=CONCAT(SEL(STATO_VENT_R,'0','1'),';');
	ADDSTRING(ADR(tempRaw), ADR(temp), tempRawLen);
	temp:=CONCAT(SEL(FILTRO,'0','1'),';');
	ADDSTRING(ADR(tempRaw), ADR(temp), tempRawLen);
	temp:=CONCAT(SEL(FLUSSO_VM,'0','1'),';');
	ADDSTRING(ADR(tempRaw), ADR(temp), tempRawLen);
	temp:=CONCAT(SEL(FLUSSO_VR,'0','1'),';');
	ADDSTRING(ADR(tempRaw), ADR(temp), tempRawLen);
	temp:=CONCAT(SEL(FILTRI_INTASATI,'0','1'),';');
	ADDSTRING(ADR(tempRaw), ADR(temp), tempRawLen);
	temp:=CONCAT(SEL(ALL_VERIFICA_VM,'0','1'),';');
	ADDSTRING(ADR(tempRaw), ADR(temp), tempRawLen);
	temp:=CONCAT(SEL(ALL_VERIFICA_VR,'0','1'),';');					(*  40 *)
	ADDSTRING(ADR(tempRaw), ADR(temp), tempRawLen);
	temp:=CONCAT(SEL(ALL_V011_MANC_SPEGN,'0','1'),';');
	ADDSTRING(ADR(tempRaw), ADR(temp), tempRawLen);
	temp:=CONCAT(SEL(ALL_V011_MANC_FUNZ,'0','1'),';');
	ADDSTRING(ADR(tempRaw), ADR(temp), tempRawLen);
	temp:=CONCAT(SEL(ALL_V012_MANC_SPEGN,'0','1'),';');
	ADDSTRING(ADR(tempRaw), ADR(temp), tempRawLen);
	temp:=CONCAT(SEL(ALL_V012_MANC_FUNZ,'0','1'),';');
	ADDSTRING(ADR(tempRaw), ADR(temp), tempRawLen);


	temp:=CONCAT(WORD_TO_STRING(Status_Log),';');
	ADDSTRING(ADR(tempRaw), ADR(temp), tempRawLen);
	temp:=CONCAT(SEL(UTA_RUN_REQ,'0','100'),';');
	ADDSTRING(ADR(tempRaw), ADR(temp), tempRawLen);
	temp:=CONCAT(SEL(UTA_STOP_REQ,'0','100'),';');
	ADDSTRING(ADR(tempRaw), ADR(temp), tempRawLen);
	temp:=CONCAT(SEL(UTA_CONTROL_MODE,'0','1'),';');
	ADDSTRING(ADR(tempRaw), ADR(temp), tempRawLen);
	temp:=(SEL(UTA_ST,'0','1'));											(*  49 *)
	ADDSTRING(ADR(tempRaw), ADR(temp), tempRawLen);


	ADDSTRING(ADR(Logger.TData), ADR(tempRaw), Logger.TLen);
END_ACTION

(* POU Plant_Objects/obj_ZTHL_01, ST *)
FUNCTION_BLOCK obj_ZTHL_01
(* === ZIGBEE AMBIENT SENSORS MT-200 ===
   v1.0[07/05/05] - Create
*)
VAR CONSTANT
	LQI_Threshold		:	WORD := 10;		(* Zigbee link quality minimum value *)
	LowBattVoltage		:	WORD := 2700;		(* Battery is considered low when reaches 1.35V each *)
END_VAR
VAR_INPUT
	(* Settings *)
	ID				: BYTE;
	Address			: BYTE;

(*	Refresh_Period	: TIME:=t#5m;
	(* Controls *)
	Refresh_Auto	: BOOL:=TRUE; (* Enable automatic refresh *)*)

	(* Modbus *)
	Refresh_Now	:	BOOL;	(* Start immediately modbus state machine *)
	retryErrMax	:	BYTE := 2;

	(* Limits *)
	Tmin			: INT := 50;
	Tmax			: INT := 400;
END_VAR
VAR_IN_OUT
	(* Interface *)
	ModBus		:obj_MODBUS;

END_VAR
VAR_OUTPUT
	(* Status *)
	Status_Log		: BYTE;
	Status_Vis 		: DWORD;
END_VAR
VAR


	state		:	INT;
	retry		:	BYTE;
	retryErr	:	BYTE;
	ReadTmr		:	TON := (PT:=T#5s);
	fModbusAlr:BOOL;


	AlarmCtr		: BYTE;
	WarningCtr		: BYTE;

	id_locale: BYTE;

	MB_RegistriLetti: ARRAY [0..20] OF INT;

